(* Logix 5000 project; controller LeakTestAuto vendor 1 type 14 code 226 rev 37.11; software revision 37.01; part 6 of 15 *)

        [78].VolumeTest.Detailed.element_data[3].result_measurement := 5.014567, [78].LeakTest.Detailed.element_data[0].result_measurement := -999.0, [79].Barcode := 'A252620460', [79].VolumeTest.UID := 25864, [79].VolumeTest.Basic.unique_id := 25864, [79].VolumeTest.Basic.channel_num := 1, [79].VolumeTest.Basic.program_num := 1, [79].VolumeTest.Basic.evaluation_code := 2, [79].VolumeTest.Basic.test_port := 1, [79].VolumeTest.Basic.year := 26, [79].VolumeTest.Basic.month := 6, [79].VolumeTest.Basic.date := 2, [79].VolumeTest.Basic.hour := 14, [79].VolumeTest.Basic.minute := 38, [79].VolumeTest.Basic.second := 3, [79].VolumeTest.Basic.flags := 12, [79].VolumeTest.Basic.Num_tests := 1, [79].VolumeTest.Basic.test_elements.test_type := 69, [79].VolumeTest.Basic.test_elements.test_eval := 2, [79].VolumeTest.Basic.test_elements.num_elements := 4, [79].VolumeTest.Detailed.unique_id := 25864, [79].VolumeTest.Detailed.num_elements := 4, [79].VolumeTest.Detailed.Test_Type := 69, [79].VolumeTest.Detailed.element_data[0].Variable_code := 245, [79].VolumeTest.Detailed.element_data[0].prec_code := 2, [79].VolumeTest.Detailed.element_data[0].Unit_code := 165, [79].VolumeTest.Detailed.element_data[0].result_measurement := 214.08073, [79].VolumeTest.Detailed.element_data[1].Variable_code := 13, [79].VolumeTest.Detailed.element_data[1].prec_code := 3, [79].VolumeTest.Detailed.element_data[1].Unit_code := 12, [79].VolumeTest.Detailed.element_data[1].result_measurement := 1.5963289, [79].VolumeTest.Detailed.element_data[2].Variable_code := 247, [79].VolumeTest.Detailed.element_data[2].prec_code := 3, [79].VolumeTest.Detailed.element_data[2].Unit_code := 12, [79].VolumeTest.Detailed.element_data[2].result_measurement := 5.013761, [79].VolumeTest.Detailed.element_data[3].Variable_code := 295, [79].VolumeTest.Detailed.element_data[3].prec_code := 3, [79].VolumeTest.Detailed.element_data[3].Unit_code := 12, [79].VolumeTest.Detailed.element_data[3].result_measurement := 5.014567, [79].LeakTest.Detailed.element_data[0].result_measurement := -999.0, [80].Barcode := 'B252620568', [80].VolumeTest.UID := 26779, [80].VolumeTest.Basic.unique_id := 26779, [80].VolumeTest.Basic.channel_num := 1, [80].VolumeTest.Basic.program_num := 1, [80].VolumeTest.Basic.evaluation_code := 1, [80].VolumeTest.Basic.test_port := 1, [80].VolumeTest.Basic.year := 26, [80].VolumeTest.Basic.month := 6, [80].VolumeTest.Basic.date := 2, [80].VolumeTest.Basic.hour := 14, [80].VolumeTest.Basic.minute := 38, [80].VolumeTest.Basic.second := 48, [80].VolumeTest.Basic.flags := 12, [80].VolumeTest.Basic.Num_tests := 1, [80].VolumeTest.Basic.test_elements.test_type := 69, [80].VolumeTest.Basic.test_elements.test_eval := 1, [80].VolumeTest.Basic.test_elements.num_elements := 4, [80].VolumeTest.Detailed.unique_id := 26779, [80].VolumeTest.Detailed.num_elements := 4,
        [80].VolumeTest.Detailed.Test_Type := 69, [80].VolumeTest.Detailed.element_data[0].Variable_code := 245, [80].VolumeTest.Detailed.element_data[0].prec_code := 2, [80].VolumeTest.Detailed.element_data[0].Unit_code := 165, [80].VolumeTest.Detailed.element_data[0].result_measurement := 185.59888, [80].VolumeTest.Detailed.element_data[1].Variable_code := 13, [80].VolumeTest.Detailed.element_data[1].prec_code := 3, [80].VolumeTest.Detailed.element_data[1].Unit_code := 12, [80].VolumeTest.Detailed.element_data[1].result_measurement := 1.7575082, [80].VolumeTest.Detailed.element_data[2].Variable_code := 247, [80].VolumeTest.Detailed.element_data[2].prec_code := 3, [80].VolumeTest.Detailed.element_data[2].Unit_code := 12, [80].VolumeTest.Detailed.element_data[2].result_measurement := 5.0194235, [80].VolumeTest.Detailed.element_data[3].Variable_code := 295, [80].VolumeTest.Detailed.element_data[3].prec_code := 3, [80].VolumeTest.Detailed.element_data[3].Unit_code := 12, [80].VolumeTest.Detailed.element_data[3].result_measurement := 5.02042, [80].LeakTest.UID := 26780, [80].LeakTest.Basic.unique_id := 26780, [80].LeakTest.Basic.channel_num := 1, [80].LeakTest.Basic.program_num := 2, [80].LeakTest.Basic.evaluation_code := 1, [80].LeakTest.Basic.test_port := 1, [80].LeakTest.Basic.year := 26, [80].LeakTest.Basic.month := 6, [80].LeakTest.Basic.date := 2, [80].LeakTest.Basic.hour := 14, [80].LeakTest.Basic.minute := 38, [80].LeakTest.Basic.second := 54, [80].LeakTest.Basic.flags := 12, [80].LeakTest.Basic.Num_tests := 1, [80].LeakTest.Basic.test_elements.test_type := 66, [80].LeakTest.Basic.test_elements.test_eval := 1, [80].LeakTest.Basic.test_elements.num_elements := 16, [80].LeakTest.Detailed.unique_id := 26780, [80].LeakTest.Detailed.num_elements := 16, [80].LeakTest.Detailed.Test_Type := 66, [80].LeakTest.Detailed.element_data[0].Variable_code := 61, [80].LeakTest.Detailed.element_data[0].prec_code := 2, [80].LeakTest.Detailed.element_data[0].Unit_code := 60, [80].LeakTest.Detailed.element_data[0].result_measurement := -0.068731606, [80].LeakTest.Detailed.element_data[1].Variable_code := 28, [80].LeakTest.Detailed.element_data[1].prec_code := 3, [80].LeakTest.Detailed.element_data[1].Unit_code := 41, [80].LeakTest.Detailed.element_data[1].result_measurement := 0.0002514571, [80].LeakTest.Detailed.element_data[2].Variable_code := 13, [80].LeakTest.Detailed.element_data[2].prec_code := 3, [80].LeakTest.Detailed.element_data[2].Unit_code := 12, [80].LeakTest.Detailed.element_data[2].result_measurement := 5.0413327, [80].LeakTest.Detailed.element_data[3].Variable_code := 75, [80].LeakTest.Detailed.element_data[3].prec_code := 2, [80].LeakTest.Detailed.element_data[3].Unit_code := 60, [80].LeakTest.Detailed.element_data[4].Variable_code := 60, [80].LeakTest.Detailed.element_data[4].prec_code := 2, [80].LeakTest.Detailed.element_data[4].Unit_code := 60, [80].LeakTest.Detailed.element_data[4].result_measurement := -0.07878989, [80].LeakTest.Detailed.element_data[5].Variable_code := 56, [80].LeakTest.Detailed.element_data[5].prec_code := 3, [80].LeakTest.Detailed.element_data[5].Unit_code := 41, [80].LeakTest.Detailed.element_data[5].result_measurement := 0.00013038516,
        [80].LeakTest.Detailed.element_data[6].Variable_code := 55, [80].LeakTest.Detailed.element_data[6].prec_code := 3, [80].LeakTest.Detailed.element_data[6].Unit_code := 12, [80].LeakTest.Detailed.element_data[6].result_measurement := 5.0413327, [80].LeakTest.Detailed.element_data[7].Variable_code := 58, [80].LeakTest.Detailed.element_data[7].prec_code := 2, [80].LeakTest.Detailed.element_data[7].Unit_code := 60, [80].LeakTest.Detailed.element_data[7].result_measurement := -1.0002404, [80].LeakTest.Detailed.element_data[8].Variable_code := 59, [80].LeakTest.Detailed.element_data[8].prec_code := 2, [80].LeakTest.Detailed.element_data[8].Unit_code := 60, [80].LeakTest.Detailed.element_data[8].result_measurement := 1.0002404, [80].LeakTest.Detailed.element_data[9].Variable_code := 12, [80].LeakTest.Detailed.element_data[9].prec_code := 3, [80].LeakTest.Detailed.element_data[9].Unit_code := 12, [80].LeakTest.Detailed.element_data[9].result_measurement := 5.000001, [80].LeakTest.Detailed.element_data[10].Variable_code := 62, [80].LeakTest.Detailed.element_data[10].prec_code := 2, [80].LeakTest.Detailed.element_data[10].Unit_code := 60, [80].LeakTest.Detailed.element_data[10].result_measurement := 1.1002644, [80].LeakTest.Detailed.element_data[11].Variable_code := 21, [80].LeakTest.Detailed.element_data[11].prec_code := 3, [80].LeakTest.Detailed.element_data[11].Unit_code := 41, [80].LeakTest.Detailed.element_data[11].result_measurement := 0.0015180558, [80].LeakTest.Detailed.element_data[12].Variable_code := 25, [80].LeakTest.Detailed.element_data[12].prec_code := 3, [80].LeakTest.Detailed.element_data[12].Unit_code := 41, [80].LeakTest.Detailed.element_data[12].result_measurement := 0.021727756, [80].LeakTest.Detailed.element_data[13].Variable_code := 216, [80].LeakTest.Detailed.element_data[13].prec_code := 3, [80].LeakTest.Detailed.element_data[13].Unit_code := 41, [80].LeakTest.Detailed.element_data[13].result_measurement := 0.00085681677, [80].LeakTest.Detailed.element_data[14].Variable_code := 218, [80].LeakTest.Detailed.element_data[14].prec_code := 3, [80].LeakTest.Detailed.element_data[14].Unit_code := 41, [80].LeakTest.Detailed.element_data[14].result_measurement := 0.01094304, [80].LeakTest.Detailed.element_data[15].Variable_code := 295, [80].LeakTest.Detailed.element_data[15].prec_code := 3, [80].LeakTest.Detailed.element_data[15].Unit_code := 12, [80].LeakTest.Detailed.element_data[15].result_measurement := 5.04273, [81].Barcode := 'B252620571', [81].VolumeTest.UID := 26782, [81].VolumeTest.Basic.unique_id := 26782, [81].VolumeTest.Basic.channel_num := 1, [81].VolumeTest.Basic.program_num := 1, [81].VolumeTest.Basic.evaluation_code := 1, [81].VolumeTest.Basic.test_port := 1, [81].VolumeTest.Basic.year := 26, [81].VolumeTest.Basic.month := 6, [81].VolumeTest.Basic.date := 2, [81].VolumeTest.Basic.hour := 14, [81].VolumeTest.Basic.minute := 39, [81].VolumeTest.Basic.second := 10, [81].VolumeTest.Basic.flags := 12, [81].VolumeTest.Basic.Num_tests := 1, [81].VolumeTest.Basic.test_elements.test_type := 69, [81].VolumeTest.Basic.test_elements.test_eval := 1, [81].VolumeTest.Basic.test_elements.num_elements := 4, [81].VolumeTest.Detailed.unique_id := 26782, [81].VolumeTest.Detailed.num_elements := 4,
        [81].VolumeTest.Detailed.Test_Type := 69, [81].VolumeTest.Detailed.element_data[0].Variable_code := 245, [81].VolumeTest.Detailed.element_data[0].prec_code := 2, [81].VolumeTest.Detailed.element_data[0].Unit_code := 165, [81].VolumeTest.Detailed.element_data[0].result_measurement := 185.52951, [81].VolumeTest.Detailed.element_data[1].Variable_code := 13, [81].VolumeTest.Detailed.element_data[1].prec_code := 3, [81].VolumeTest.Detailed.element_data[1].Unit_code := 12, [81].VolumeTest.Detailed.element_data[1].result_measurement := 1.757997, [81].VolumeTest.Detailed.element_data[2].Variable_code := 247, [81].VolumeTest.Detailed.element_data[2].prec_code := 3, [81].VolumeTest.Detailed.element_data[2].Unit_code := 12, [81].VolumeTest.Detailed.element_data[2].result_measurement := 5.0196004, [81].VolumeTest.Detailed.element_data[3].Variable_code := 295, [81].VolumeTest.Detailed.element_data[3].prec_code := 3, [81].VolumeTest.Detailed.element_data[3].Unit_code := 12, [81].VolumeTest.Detailed.element_data[3].result_measurement := 5.0203876, [81].LeakTest.UID := 26783, [81].LeakTest.Basic.unique_id := 26783, [81].LeakTest.Basic.channel_num := 1, [81].LeakTest.Basic.program_num := 2, [81].LeakTest.Basic.evaluation_code := 1, [81].LeakTest.Basic.test_port := 1, [81].LeakTest.Basic.year := 26, [81].LeakTest.Basic.month := 6, [81].LeakTest.Basic.date := 2, [81].LeakTest.Basic.hour := 14, [81].LeakTest.Basic.minute := 39, [81].LeakTest.Basic.second := 17, [81].LeakTest.Basic.flags := 12, [81].LeakTest.Basic.Num_tests := 1, [81].LeakTest.Basic.test_elements.test_type := 66, [81].LeakTest.Basic.test_elements.test_eval := 1, [81].LeakTest.Basic.test_elements.num_elements := 16, [81].LeakTest.Detailed.unique_id := 26783, [81].LeakTest.Detailed.num_elements := 16, [81].LeakTest.Detailed.Test_Type := 66, [81].LeakTest.Detailed.element_data[0].Variable_code := 61, [81].LeakTest.Detailed.element_data[0].prec_code := 2, [81].LeakTest.Detailed.element_data[0].Unit_code := 60, [81].LeakTest.Detailed.element_data[0].result_measurement := -0.059232116, [81].LeakTest.Detailed.element_data[1].Variable_code := 28, [81].LeakTest.Detailed.element_data[1].prec_code := 3, [81].LeakTest.Detailed.element_data[1].Unit_code := 41, [81].LeakTest.Detailed.element_data[1].result_measurement := 0.00042840838, [81].LeakTest.Detailed.element_data[2].Variable_code := 13, [81].LeakTest.Detailed.element_data[2].prec_code := 3, [81].LeakTest.Detailed.element_data[2].Unit_code := 12, [81].LeakTest.Detailed.element_data[2].result_measurement := 5.040425, [81].LeakTest.Detailed.element_data[3].Variable_code := 75, [81].LeakTest.Detailed.element_data[3].prec_code := 2, [81].LeakTest.Detailed.element_data[3].Unit_code := 60, [81].LeakTest.Detailed.element_data[4].Variable_code := 60, [81].LeakTest.Detailed.element_data[4].prec_code := 2, [81].LeakTest.Detailed.element_data[4].Unit_code := 60, [81].LeakTest.Detailed.element_data[4].result_measurement := -0.068731606, [81].LeakTest.Detailed.element_data[5].Variable_code := 56, [81].LeakTest.Detailed.element_data[5].prec_code := 3, [81].LeakTest.Detailed.element_data[5].Unit_code := 41, [81].LeakTest.Detailed.element_data[5].result_measurement := 0.00022351742,
        [81].LeakTest.Detailed.element_data[6].Variable_code := 55, [81].LeakTest.Detailed.element_data[6].prec_code := 3, [81].LeakTest.Detailed.element_data[6].Unit_code := 12, [81].LeakTest.Detailed.element_data[6].result_measurement := 5.040425, [81].LeakTest.Detailed.element_data[7].Variable_code := 58, [81].LeakTest.Detailed.element_data[7].prec_code := 2, [81].LeakTest.Detailed.element_data[7].Unit_code := 60, [81].LeakTest.Detailed.element_data[7].result_measurement := -1.0002404, [81].LeakTest.Detailed.element_data[8].Variable_code := 59, [81].LeakTest.Detailed.element_data[8].prec_code := 2, [81].LeakTest.Detailed.element_data[8].Unit_code := 60, [81].LeakTest.Detailed.element_data[8].result_measurement := 1.0002404, [81].LeakTest.Detailed.element_data[9].Variable_code := 12, [81].LeakTest.Detailed.element_data[9].prec_code := 3, [81].LeakTest.Detailed.element_data[9].Unit_code := 12, [81].LeakTest.Detailed.element_data[9].result_measurement := 5.000001, [81].LeakTest.Detailed.element_data[10].Variable_code := 62, [81].LeakTest.Detailed.element_data[10].prec_code := 2, [81].LeakTest.Detailed.element_data[10].Unit_code := 60, [81].LeakTest.Detailed.element_data[10].result_measurement := 1.1002644, [81].LeakTest.Detailed.element_data[11].Variable_code := 21, [81].LeakTest.Detailed.element_data[11].prec_code := 3, [81].LeakTest.Detailed.element_data[11].Unit_code := 41, [81].LeakTest.Detailed.element_data[11].result_measurement := 0.0015180558, [81].LeakTest.Detailed.element_data[12].Variable_code := 25, [81].LeakTest.Detailed.element_data[12].prec_code := 3, [81].LeakTest.Detailed.element_data[12].Unit_code := 41, [81].LeakTest.Detailed.element_data[12].result_measurement := 0.021727756, [81].LeakTest.Detailed.element_data[13].Variable_code := 216, [81].LeakTest.Detailed.element_data[13].prec_code := 3, [81].LeakTest.Detailed.element_data[13].Unit_code := 41, [81].LeakTest.Detailed.element_data[13].result_measurement := 0.00085681677, [81].LeakTest.Detailed.element_data[14].Variable_code := 218, [81].LeakTest.Detailed.element_data[14].prec_code := 3, [81].LeakTest.Detailed.element_data[14].Unit_code := 41, [81].LeakTest.Detailed.element_data[14].result_measurement := 0.01094304, [81].LeakTest.Detailed.element_data[15].Variable_code := 295, [81].LeakTest.Detailed.element_data[15].prec_code := 3, [81].LeakTest.Detailed.element_data[15].Unit_code := 12, [81].LeakTest.Detailed.element_data[15].result_measurement := 5.0419664, [82].Barcode := 'B252620555', [82].VolumeTest.UID := 25866, [82].VolumeTest.Basic.unique_id := 25866, [82].VolumeTest.Basic.channel_num := 1, [82].VolumeTest.Basic.program_num := 1, [82].VolumeTest.Basic.evaluation_code := 1, [82].VolumeTest.Basic.test_port := 1, [82].VolumeTest.Basic.year := 26, [82].VolumeTest.Basic.month := 6, [82].VolumeTest.Basic.date := 2, [82].VolumeTest.Basic.hour := 14, [82].VolumeTest.Basic.minute := 38, [82].VolumeTest.Basic.second := 25, [82].VolumeTest.Basic.flags := 12, [82].VolumeTest.Basic.Num_tests := 1, [82].VolumeTest.Basic.test_elements.test_type := 69, [82].VolumeTest.Basic.test_elements.test_eval := 1, [82].VolumeTest.Basic.test_elements.num_elements := 4, [82].VolumeTest.Detailed.unique_id := 25866, [82].VolumeTest.Detailed.num_elements := 4,
        [82].VolumeTest.Detailed.Test_Type := 69, [82].VolumeTest.Detailed.element_data[0].Variable_code := 245, [82].VolumeTest.Detailed.element_data[0].prec_code := 2, [82].VolumeTest.Detailed.element_data[0].Unit_code := 165, [82].VolumeTest.Detailed.element_data[0].result_measurement := 188.30235, [82].VolumeTest.Detailed.element_data[1].Variable_code := 13, [82].VolumeTest.Detailed.element_data[1].prec_code := 3, [82].VolumeTest.Detailed.element_data[1].Unit_code := 12, [82].VolumeTest.Detailed.element_data[1].result_measurement := 1.7390168, [82].VolumeTest.Detailed.element_data[2].Variable_code := 247, [82].VolumeTest.Detailed.element_data[2].prec_code := 3, [82].VolumeTest.Detailed.element_data[2].Unit_code := 12, [82].VolumeTest.Detailed.element_data[2].result_measurement := 5.013626, [82].VolumeTest.Detailed.element_data[3].Variable_code := 295, [82].VolumeTest.Detailed.element_data[3].prec_code := 3, [82].VolumeTest.Detailed.element_data[3].Unit_code := 12, [82].VolumeTest.Detailed.element_data[3].result_measurement := 5.0143385, [82].LeakTest.UID := 25867, [82].LeakTest.Basic.unique_id := 25867, [82].LeakTest.Basic.channel_num := 1, [82].LeakTest.Basic.program_num := 2, [82].LeakTest.Basic.evaluation_code := 1, [82].LeakTest.Basic.test_port := 1, [82].LeakTest.Basic.year := 26, [82].LeakTest.Basic.month := 6, [82].LeakTest.Basic.date := 2, [82].LeakTest.Basic.hour := 14, [82].LeakTest.Basic.minute := 38, [82].LeakTest.Basic.second := 32, [82].LeakTest.Basic.flags := 12, [82].LeakTest.Basic.Num_tests := 1, [82].LeakTest.Basic.test_elements.test_type := 66, [82].LeakTest.Basic.test_elements.test_eval := 1, [82].LeakTest.Basic.test_elements.num_elements := 16, [82].LeakTest.Detailed.unique_id := 25867, [82].LeakTest.Detailed.num_elements := 16, [82].LeakTest.Detailed.Test_Type := 66, [82].LeakTest.Detailed.element_data[0].Variable_code := 61, [82].LeakTest.Detailed.element_data[0].prec_code := 2, [82].LeakTest.Detailed.element_data[0].Unit_code := 60, [82].LeakTest.Detailed.element_data[0].result_measurement := -0.05811453, [82].LeakTest.Detailed.element_data[1].Variable_code := 28, [82].LeakTest.Detailed.element_data[1].prec_code := 3, [82].LeakTest.Detailed.element_data[1].Unit_code := 41, [82].LeakTest.Detailed.element_data[1].result_measurement := 0.00045634806, [82].LeakTest.Detailed.element_data[2].Variable_code := 13, [82].LeakTest.Detailed.element_data[2].prec_code := 3, [82].LeakTest.Detailed.element_data[2].Unit_code := 12, [82].LeakTest.Detailed.element_data[2].result_measurement := 5.033845, [82].LeakTest.Detailed.element_data[3].Variable_code := 75, [82].LeakTest.Detailed.element_data[3].prec_code := 2, [82].LeakTest.Detailed.element_data[3].Unit_code := 60, [82].LeakTest.Detailed.element_data[4].Variable_code := 60, [82].LeakTest.Detailed.element_data[4].prec_code := 2, [82].LeakTest.Detailed.element_data[4].Unit_code := 60, [82].LeakTest.Detailed.element_data[4].result_measurement := -0.07431954, [82].LeakTest.Detailed.element_data[5].Variable_code := 56, [82].LeakTest.Detailed.element_data[5].prec_code := 3, [82].LeakTest.Detailed.element_data[5].Unit_code := 41, [82].LeakTest.Detailed.element_data[5].result_measurement := 0.00017695129,
        [82].LeakTest.Detailed.element_data[6].Variable_code := 55, [82].LeakTest.Detailed.element_data[6].prec_code := 3, [82].LeakTest.Detailed.element_data[6].Unit_code := 12, [82].LeakTest.Detailed.element_data[6].result_measurement := 5.033845, [82].LeakTest.Detailed.element_data[7].Variable_code := 58, [82].LeakTest.Detailed.element_data[7].prec_code := 2, [82].LeakTest.Detailed.element_data[7].Unit_code := 60, [82].LeakTest.Detailed.element_data[7].result_measurement := -1.0002404, [82].LeakTest.Detailed.element_data[8].Variable_code := 59, [82].LeakTest.Detailed.element_data[8].prec_code := 2, [82].LeakTest.Detailed.element_data[8].Unit_code := 60, [82].LeakTest.Detailed.element_data[8].result_measurement := 1.0002404, [82].LeakTest.Detailed.element_data[9].Variable_code := 12, [82].LeakTest.Detailed.element_data[9].prec_code := 3, [82].LeakTest.Detailed.element_data[9].Unit_code := 12, [82].LeakTest.Detailed.element_data[9].result_measurement := 5.000001, [82].LeakTest.Detailed.element_data[10].Variable_code := 62, [82].LeakTest.Detailed.element_data[10].prec_code := 2, [82].LeakTest.Detailed.element_data[10].Unit_code := 60, [82].LeakTest.Detailed.element_data[10].result_measurement := 1.109764, [82].LeakTest.Detailed.element_data[11].Variable_code := 21, [82].LeakTest.Detailed.element_data[11].prec_code := 3, [82].LeakTest.Detailed.element_data[11].Unit_code := 41, [82].LeakTest.Detailed.element_data[11].result_measurement := 0.0015180558, [82].LeakTest.Detailed.element_data[12].Variable_code := 25, [82].LeakTest.Detailed.element_data[12].prec_code := 3, [82].LeakTest.Detailed.element_data[12].Unit_code := 41, [82].LeakTest.Detailed.element_data[12].result_measurement := 0.021727756, [82].LeakTest.Detailed.element_data[13].Variable_code := 216, [82].LeakTest.Detailed.element_data[13].prec_code := 3, [82].LeakTest.Detailed.element_data[13].Unit_code := 41, [82].LeakTest.Detailed.element_data[13].result_measurement := 0.00085681677, [82].LeakTest.Detailed.element_data[14].Variable_code := 218, [82].LeakTest.Detailed.element_data[14].prec_code := 3, [82].LeakTest.Detailed.element_data[14].Unit_code := 41, [82].LeakTest.Detailed.element_data[14].result_measurement := 0.01094304, [82].LeakTest.Detailed.element_data[15].Variable_code := 295, [82].LeakTest.Detailed.element_data[15].prec_code := 3, [82].LeakTest.Detailed.element_data[15].Unit_code := 12, [82].LeakTest.Detailed.element_data[15].result_measurement := 5.03602, [83].Barcode := 'B252620555', [83].VolumeTest.UID := 41945, [83].VolumeTest.Basic.unique_id := 41945, [83].VolumeTest.Basic.channel_num := 1, [83].VolumeTest.Basic.program_num := 1, [83].VolumeTest.Basic.evaluation_code := 1, [83].VolumeTest.Basic.test_port := 1, [83].VolumeTest.Basic.year := 26, [83].VolumeTest.Basic.month := 6, [83].VolumeTest.Basic.date := 4, [83].VolumeTest.Basic.hour := 12, [83].VolumeTest.Basic.minute := 27, [83].VolumeTest.Basic.second := 3, [83].VolumeTest.Basic.flags := 12, [83].VolumeTest.Basic.Num_tests := 1, [83].VolumeTest.Basic.test_elements.test_type := 69, [83].VolumeTest.Basic.test_elements.test_eval := 1, [83].VolumeTest.Basic.test_elements.num_elements := 4, [83].VolumeTest.Detailed.unique_id := 41945, [83].VolumeTest.Detailed.num_elements := 4,
        [83].VolumeTest.Detailed.Test_Type := 69, [83].VolumeTest.Detailed.element_data[0].Variable_code := 245, [83].VolumeTest.Detailed.element_data[0].prec_code := 2, [83].VolumeTest.Detailed.element_data[0].Unit_code := 165, [83].VolumeTest.Detailed.element_data[0].result_measurement := 186.67934, [83].VolumeTest.Detailed.element_data[1].Variable_code := 13, [83].VolumeTest.Detailed.element_data[1].prec_code := 3, [83].VolumeTest.Detailed.element_data[1].Unit_code := 12, [83].VolumeTest.Detailed.element_data[1].result_measurement := 1.7815549, [83].VolumeTest.Detailed.element_data[2].Variable_code := 247, [83].VolumeTest.Detailed.element_data[2].prec_code := 3, [83].VolumeTest.Detailed.element_data[2].Unit_code := 12, [83].VolumeTest.Detailed.element_data[2].result_measurement := 5.10735, [83].VolumeTest.Detailed.element_data[3].Variable_code := 295, [83].VolumeTest.Detailed.element_data[3].prec_code := 3, [83].VolumeTest.Detailed.element_data[3].Unit_code := 12, [83].VolumeTest.Detailed.element_data[3].result_measurement := 5.107876, [83].LeakTest.UID := 41946, [83].LeakTest.Basic.unique_id := 41946, [83].LeakTest.Basic.channel_num := 1, [83].LeakTest.Basic.program_num := 2, [83].LeakTest.Basic.evaluation_code := 1, [83].LeakTest.Basic.test_port := 1, [83].LeakTest.Basic.year := 26, [83].LeakTest.Basic.month := 6, [83].LeakTest.Basic.date := 4, [83].LeakTest.Basic.hour := 12, [83].LeakTest.Basic.minute := 27, [83].LeakTest.Basic.second := 10, [83].LeakTest.Basic.flags := 12, [83].LeakTest.Basic.Num_tests := 1, [83].LeakTest.Basic.test_elements.test_type := 66, [83].LeakTest.Basic.test_elements.test_eval := 1, [83].LeakTest.Basic.test_elements.num_elements := 16, [83].LeakTest.Detailed.unique_id := 41946, [83].LeakTest.Detailed.num_elements := 16, [83].LeakTest.Detailed.Test_Type := 66, [83].LeakTest.Detailed.element_data[0].Variable_code := 61, [83].LeakTest.Detailed.element_data[0].prec_code := 2, [83].LeakTest.Detailed.element_data[0].Unit_code := 60, [83].LeakTest.Detailed.element_data[0].result_measurement := -0.07431954, [83].LeakTest.Detailed.element_data[1].Variable_code := 28, [83].LeakTest.Detailed.element_data[1].prec_code := 3, [83].LeakTest.Detailed.element_data[1].Unit_code := 41, [83].LeakTest.Detailed.element_data[1].result_measurement := 0.00014901161, [83].LeakTest.Detailed.element_data[2].Variable_code := 13, [83].LeakTest.Detailed.element_data[2].prec_code := 3, [83].LeakTest.Detailed.element_data[2].Unit_code := 12, [83].LeakTest.Detailed.element_data[2].result_measurement := 5.137217, [83].LeakTest.Detailed.element_data[3].Variable_code := 75, [83].LeakTest.Detailed.element_data[3].prec_code := 2, [83].LeakTest.Detailed.element_data[3].Unit_code := 60, [83].LeakTest.Detailed.element_data[4].Variable_code := 60, [83].LeakTest.Detailed.element_data[4].prec_code := 2, [83].LeakTest.Detailed.element_data[4].Unit_code := 60, [83].LeakTest.Detailed.element_data[4].result_measurement := -0.08214265, [83].LeakTest.Detailed.element_data[5].Variable_code := 56, [83].LeakTest.Detailed.element_data[5].prec_code := 3, [83].LeakTest.Detailed.element_data[5].Unit_code := 41, [83].LeakTest.Detailed.element_data[5].result_measurement := 0.00010244548,
        [83].LeakTest.Detailed.element_data[6].Variable_code := 55, [83].LeakTest.Detailed.element_data[6].prec_code := 3, [83].LeakTest.Detailed.element_data[6].Unit_code := 12, [83].LeakTest.Detailed.element_data[6].result_measurement := 5.137217, [83].LeakTest.Detailed.element_data[7].Variable_code := 58, [83].LeakTest.Detailed.element_data[7].prec_code := 2, [83].LeakTest.Detailed.element_data[7].Unit_code := 60, [83].LeakTest.Detailed.element_data[7].result_measurement := -1.0002404, [83].LeakTest.Detailed.element_data[8].Variable_code := 59, [83].LeakTest.Detailed.element_data[8].prec_code := 2, [83].LeakTest.Detailed.element_data[8].Unit_code := 60, [83].LeakTest.Detailed.element_data[8].result_measurement := 1.0002404, [83].LeakTest.Detailed.element_data[9].Variable_code := 12, [83].LeakTest.Detailed.element_data[9].prec_code := 3, [83].LeakTest.Detailed.element_data[9].Unit_code := 12, [83].LeakTest.Detailed.element_data[9].result_measurement := 5.000001, [83].LeakTest.Detailed.element_data[10].Variable_code := 62, [83].LeakTest.Detailed.element_data[10].prec_code := 2, [83].LeakTest.Detailed.element_data[10].Unit_code := 60, [83].LeakTest.Detailed.element_data[10].result_measurement := 1.1002644, [83].LeakTest.Detailed.element_data[11].Variable_code := 21, [83].LeakTest.Detailed.element_data[11].prec_code := 3, [83].LeakTest.Detailed.element_data[11].Unit_code := 41, [83].LeakTest.Detailed.element_data[11].result_measurement := 0.0015180558, [83].LeakTest.Detailed.element_data[12].Variable_code := 25, [83].LeakTest.Detailed.element_data[12].prec_code := 3, [83].LeakTest.Detailed.element_data[12].Unit_code := 41, [83].LeakTest.Detailed.element_data[12].result_measurement := 0.021727756, [83].LeakTest.Detailed.element_data[13].Variable_code := 216, [83].LeakTest.Detailed.element_data[13].prec_code := 3, [83].LeakTest.Detailed.element_data[13].Unit_code := 41, [83].LeakTest.Detailed.element_data[13].result_measurement := 0.00085681677, [83].LeakTest.Detailed.element_data[14].Variable_code := 218, [83].LeakTest.Detailed.element_data[14].prec_code := 3, [83].LeakTest.Detailed.element_data[14].Unit_code := 41, [83].LeakTest.Detailed.element_data[14].result_measurement := 0.01094304, [83].LeakTest.Detailed.element_data[15].Variable_code := 295, [83].LeakTest.Detailed.element_data[15].prec_code := 3, [83].LeakTest.Detailed.element_data[15].Unit_code := 12, [83].LeakTest.Detailed.element_data[15].result_measurement := 5.1387258, [84].Barcode := 'B252620571', [84].VolumeTest.UID := 42936, [84].VolumeTest.Basic.unique_id := 42936, [84].VolumeTest.Basic.channel_num := 1, [84].VolumeTest.Basic.program_num := 1, [84].VolumeTest.Basic.evaluation_code := 1, [84].VolumeTest.Basic.test_port := 1, [84].VolumeTest.Basic.year := 26, [84].VolumeTest.Basic.month := 6, [84].VolumeTest.Basic.date := 4, [84].VolumeTest.Basic.hour := 12, [84].VolumeTest.Basic.minute := 27, [84].VolumeTest.Basic.second := 27, [84].VolumeTest.Basic.flags := 12, [84].VolumeTest.Basic.Num_tests := 1, [84].VolumeTest.Basic.test_elements.test_type := 69, [84].VolumeTest.Basic.test_elements.test_eval := 1, [84].VolumeTest.Basic.test_elements.num_elements := 4, [84].VolumeTest.Detailed.unique_id := 42936, [84].VolumeTest.Detailed.num_elements := 4,
        [84].VolumeTest.Detailed.Test_Type := 69, [84].VolumeTest.Detailed.element_data[0].Variable_code := 245, [84].VolumeTest.Detailed.element_data[0].prec_code := 2, [84].VolumeTest.Detailed.element_data[0].Unit_code := 165, [84].VolumeTest.Detailed.element_data[0].result_measurement := 188.14069, [84].VolumeTest.Detailed.element_data[1].Variable_code := 13, [84].VolumeTest.Detailed.element_data[1].prec_code := 3, [84].VolumeTest.Detailed.element_data[1].Unit_code := 12, [84].VolumeTest.Detailed.element_data[1].result_measurement := 1.8124143, [84].VolumeTest.Detailed.element_data[2].Variable_code := 247, [84].VolumeTest.Detailed.element_data[2].prec_code := 3, [84].VolumeTest.Detailed.element_data[2].Unit_code := 12, [84].VolumeTest.Detailed.element_data[2].result_measurement := 5.222303, [84].VolumeTest.Detailed.element_data[3].Variable_code := 295, [84].VolumeTest.Detailed.element_data[3].prec_code := 3, [84].VolumeTest.Detailed.element_data[3].Unit_code := 12, [84].VolumeTest.Detailed.element_data[3].result_measurement := 5.224529, [84].LeakTest.UID := 42937, [84].LeakTest.Basic.unique_id := 42937, [84].LeakTest.Basic.channel_num := 1, [84].LeakTest.Basic.program_num := 2, [84].LeakTest.Basic.evaluation_code := 1, [84].LeakTest.Basic.test_port := 1, [84].LeakTest.Basic.year := 26, [84].LeakTest.Basic.month := 6, [84].LeakTest.Basic.date := 4, [84].LeakTest.Basic.hour := 12, [84].LeakTest.Basic.minute := 27, [84].LeakTest.Basic.second := 33, [84].LeakTest.Basic.flags := 12, [84].LeakTest.Basic.Num_tests := 1, [84].LeakTest.Basic.test_elements.test_type := 66, [84].LeakTest.Basic.test_elements.test_eval := 1, [84].LeakTest.Basic.test_elements.num_elements := 16, [84].LeakTest.Detailed.unique_id := 42937, [84].LeakTest.Detailed.num_elements := 16, [84].LeakTest.Detailed.Test_Type := 66, [84].LeakTest.Detailed.element_data[0].Variable_code := 61, [84].LeakTest.Detailed.element_data[0].prec_code := 2, [84].LeakTest.Detailed.element_data[0].Unit_code := 60, [84].LeakTest.Detailed.element_data[0].result_measurement := -0.005029142, [84].LeakTest.Detailed.element_data[1].Variable_code := 28, [84].LeakTest.Detailed.element_data[1].prec_code := 3, [84].LeakTest.Detailed.element_data[1].Unit_code := 41, [84].LeakTest.Detailed.element_data[1].result_measurement := -0.00010244548, [84].LeakTest.Detailed.element_data[2].Variable_code := 13, [84].LeakTest.Detailed.element_data[2].prec_code := 3, [84].LeakTest.Detailed.element_data[2].Unit_code := 12, [84].LeakTest.Detailed.element_data[2].result_measurement := 5.2362356, [84].LeakTest.Detailed.element_data[3].Variable_code := 75, [84].LeakTest.Detailed.element_data[3].prec_code := 2, [84].LeakTest.Detailed.element_data[3].Unit_code := 60, [84].LeakTest.Detailed.element_data[4].Variable_code := 60, [84].LeakTest.Detailed.element_data[4].prec_code := 2, [84].LeakTest.Detailed.element_data[4].Unit_code := 60, [84].LeakTest.Detailed.element_data[4].result_measurement := -0.022910535, [84].LeakTest.Detailed.element_data[5].Variable_code := 56, [84].LeakTest.Detailed.element_data[5].prec_code := 3, [84].LeakTest.Detailed.element_data[5].Unit_code := 41, [84].LeakTest.Detailed.element_data[5].result_measurement := -0.00027474016,
        [84].LeakTest.Detailed.element_data[6].Variable_code := 55, [84].LeakTest.Detailed.element_data[6].prec_code := 3, [84].LeakTest.Detailed.element_data[6].Unit_code := 12, [84].LeakTest.Detailed.element_data[6].result_measurement := 5.2362356, [84].LeakTest.Detailed.element_data[7].Variable_code := 58, [84].LeakTest.Detailed.element_data[7].prec_code := 2, [84].LeakTest.Detailed.element_data[7].Unit_code := 60, [84].LeakTest.Detailed.element_data[7].result_measurement := -1.0002404, [84].LeakTest.Detailed.element_data[8].Variable_code := 59, [84].LeakTest.Detailed.element_data[8].prec_code := 2, [84].LeakTest.Detailed.element_data[8].Unit_code := 60, [84].LeakTest.Detailed.element_data[8].result_measurement := 1.0002404, [84].LeakTest.Detailed.element_data[9].Variable_code := 12, [84].LeakTest.Detailed.element_data[9].prec_code := 3, [84].LeakTest.Detailed.element_data[9].Unit_code := 12, [84].LeakTest.Detailed.element_data[9].result_measurement := 5.000001, [84].LeakTest.Detailed.element_data[10].Variable_code := 62, [84].LeakTest.Detailed.element_data[10].prec_code := 2, [84].LeakTest.Detailed.element_data[10].Unit_code := 60, [84].LeakTest.Detailed.element_data[10].result_measurement := 1.1298805, [84].LeakTest.Detailed.element_data[11].Variable_code := 21, [84].LeakTest.Detailed.element_data[11].prec_code := 3, [84].LeakTest.Detailed.element_data[11].Unit_code := 41, [84].LeakTest.Detailed.element_data[11].result_measurement := 4.656613e-06, [84].LeakTest.Detailed.element_data[12].Variable_code := 25, [84].LeakTest.Detailed.element_data[12].prec_code := 3, [84].LeakTest.Detailed.element_data[12].Unit_code := 41, [84].LeakTest.Detailed.element_data[12].result_measurement := 0.023245811, [84].LeakTest.Detailed.element_data[13].Variable_code := 216, [84].LeakTest.Detailed.element_data[13].prec_code := 3, [84].LeakTest.Detailed.element_data[13].Unit_code := 41, [84].LeakTest.Detailed.element_data[13].result_measurement := -3.7252903e-05, [84].LeakTest.Detailed.element_data[14].Variable_code := 218, [84].LeakTest.Detailed.element_data[14].prec_code := 3, [84].LeakTest.Detailed.element_data[14].Unit_code := 41, [84].LeakTest.Detailed.element_data[14].result_measurement := 0.011632219, [84].LeakTest.Detailed.element_data[15].Variable_code := 295, [84].LeakTest.Detailed.element_data[15].prec_code := 3, [84].LeakTest.Detailed.element_data[15].Unit_code := 12, [84].LeakTest.Detailed.element_data[15].result_measurement := 5.237949, [85].Barcode := 'B252620865', [85].VolumeTest.UID := 42939, [85].VolumeTest.Basic.unique_id := 42939, [85].VolumeTest.Basic.channel_num := 1, [85].VolumeTest.Basic.program_num := 1, [85].VolumeTest.Basic.evaluation_code := 1, [85].VolumeTest.Basic.test_port := 1, [85].VolumeTest.Basic.year := 26, [85].VolumeTest.Basic.month := 6, [85].VolumeTest.Basic.date := 4, [85].VolumeTest.Basic.hour := 12, [85].VolumeTest.Basic.minute := 28, [85].VolumeTest.Basic.second := 27, [85].VolumeTest.Basic.flags := 12, [85].VolumeTest.Basic.Num_tests := 1, [85].VolumeTest.Basic.test_elements.test_type := 69, [85].VolumeTest.Basic.test_elements.test_eval := 1, [85].VolumeTest.Basic.test_elements.num_elements := 4, [85].VolumeTest.Detailed.unique_id := 42939, [85].VolumeTest.Detailed.num_elements := 4,
        [85].VolumeTest.Detailed.Test_Type := 69, [85].VolumeTest.Detailed.element_data[0].Variable_code := 245, [85].VolumeTest.Detailed.element_data[0].prec_code := 2, [85].VolumeTest.Detailed.element_data[0].Unit_code := 165, [85].VolumeTest.Detailed.element_data[0].result_measurement := 188.86253, [85].VolumeTest.Detailed.element_data[1].Variable_code := 13, [85].VolumeTest.Detailed.element_data[1].prec_code := 3, [85].VolumeTest.Detailed.element_data[1].Unit_code := 12, [85].VolumeTest.Detailed.element_data[1].result_measurement := 1.8058717, [85].VolumeTest.Detailed.element_data[2].Variable_code := 247, [85].VolumeTest.Detailed.element_data[2].prec_code := 3, [85].VolumeTest.Detailed.element_data[2].Unit_code := 12, [85].VolumeTest.Detailed.element_data[2].result_measurement := 5.216487, [85].VolumeTest.Detailed.element_data[3].Variable_code := 295, [85].VolumeTest.Detailed.element_data[3].prec_code := 3, [85].VolumeTest.Detailed.element_data[3].Unit_code := 12, [85].VolumeTest.Detailed.element_data[3].result_measurement := 5.2191176, [85].LeakTest.UID := 42940, [85].LeakTest.Basic.unique_id := 42940, [85].LeakTest.Basic.channel_num := 1, [85].LeakTest.Basic.program_num := 2, [85].LeakTest.Basic.evaluation_code := 1, [85].LeakTest.Basic.test_port := 1, [85].LeakTest.Basic.year := 26, [85].LeakTest.Basic.month := 6, [85].LeakTest.Basic.date := 4, [85].LeakTest.Basic.hour := 12, [85].LeakTest.Basic.minute := 28, [85].LeakTest.Basic.second := 34, [85].LeakTest.Basic.flags := 12, [85].LeakTest.Basic.Num_tests := 1, [85].LeakTest.Basic.test_elements.test_type := 66, [85].LeakTest.Basic.test_elements.test_eval := 1, [85].LeakTest.Basic.test_elements.num_elements := 16, [85].LeakTest.Detailed.unique_id := 42940, [85].LeakTest.Detailed.num_elements := 16, [85].LeakTest.Detailed.Test_Type := 66, [85].LeakTest.Detailed.element_data[0].Variable_code := 61, [85].LeakTest.Detailed.element_data[0].prec_code := 2, [85].LeakTest.Detailed.element_data[0].Unit_code := 60, [85].LeakTest.Detailed.element_data[0].result_measurement := -0.0067055225, [85].LeakTest.Detailed.element_data[1].Variable_code := 28, [85].LeakTest.Detailed.element_data[1].prec_code := 3, [85].LeakTest.Detailed.element_data[1].Unit_code := 41, [85].LeakTest.Detailed.element_data[1].result_measurement := -0.00013969839, [85].LeakTest.Detailed.element_data[2].Variable_code := 13, [85].LeakTest.Detailed.element_data[2].prec_code := 3, [85].LeakTest.Detailed.element_data[2].Unit_code := 12, [85].LeakTest.Detailed.element_data[2].result_measurement := 5.2345915, [85].LeakTest.Detailed.element_data[3].Variable_code := 75, [85].LeakTest.Detailed.element_data[3].prec_code := 2, [85].LeakTest.Detailed.element_data[3].Unit_code := 60, [85].LeakTest.Detailed.element_data[4].Variable_code := 60, [85].LeakTest.Detailed.element_data[4].prec_code := 2, [85].LeakTest.Detailed.element_data[4].Unit_code := 60, [85].LeakTest.Detailed.element_data[4].result_measurement := -0.0044703484, [85].LeakTest.Detailed.element_data[5].Variable_code := 56, [85].LeakTest.Detailed.element_data[5].prec_code := 3, [85].LeakTest.Detailed.element_data[5].Unit_code := 41, [85].LeakTest.Detailed.element_data[5].result_measurement := -8.8475645e-05,
        [85].LeakTest.Detailed.element_data[6].Variable_code := 55, [85].LeakTest.Detailed.element_data[6].prec_code := 3, [85].LeakTest.Detailed.element_data[6].Unit_code := 12, [85].LeakTest.Detailed.element_data[6].result_measurement := 5.2345915, [85].LeakTest.Detailed.element_data[7].Variable_code := 58, [85].LeakTest.Detailed.element_data[7].prec_code := 2, [85].LeakTest.Detailed.element_data[7].Unit_code := 60, [85].LeakTest.Detailed.element_data[7].result_measurement := -1.0002404, [85].LeakTest.Detailed.element_data[8].Variable_code := 59, [85].LeakTest.Detailed.element_data[8].prec_code := 2, [85].LeakTest.Detailed.element_data[8].Unit_code := 60, [85].LeakTest.Detailed.element_data[8].result_measurement := 1.0002404, [85].LeakTest.Detailed.element_data[9].Variable_code := 12, [85].LeakTest.Detailed.element_data[9].prec_code := 3, [85].LeakTest.Detailed.element_data[9].Unit_code := 12, [85].LeakTest.Detailed.element_data[9].result_measurement := 5.000001, [85].LeakTest.Detailed.element_data[10].Variable_code := 62, [85].LeakTest.Detailed.element_data[10].prec_code := 2, [85].LeakTest.Detailed.element_data[10].Unit_code := 60, [85].LeakTest.Detailed.element_data[10].result_measurement := 1.1298805, [85].LeakTest.Detailed.element_data[11].Variable_code := 21, [85].LeakTest.Detailed.element_data[11].prec_code := 3, [85].LeakTest.Detailed.element_data[11].Unit_code := 41, [85].LeakTest.Detailed.element_data[11].result_measurement := 4.656613e-06, [85].LeakTest.Detailed.element_data[12].Variable_code := 25, [85].LeakTest.Detailed.element_data[12].prec_code := 3, [85].LeakTest.Detailed.element_data[12].Unit_code := 41, [85].LeakTest.Detailed.element_data[12].result_measurement := 0.023245811, [85].LeakTest.Detailed.element_data[13].Variable_code := 216, [85].LeakTest.Detailed.element_data[13].prec_code := 3, [85].LeakTest.Detailed.element_data[13].Unit_code := 41, [85].LeakTest.Detailed.element_data[13].result_measurement := -3.7252903e-05, [85].LeakTest.Detailed.element_data[14].Variable_code := 218, [85].LeakTest.Detailed.element_data[14].prec_code := 3, [85].LeakTest.Detailed.element_data[14].Unit_code := 41, [85].LeakTest.Detailed.element_data[14].result_measurement := 0.011632219, [85].LeakTest.Detailed.element_data[15].Variable_code := 295, [85].LeakTest.Detailed.element_data[15].prec_code := 3, [85].LeakTest.Detailed.element_data[15].Unit_code := 12, [85].LeakTest.Detailed.element_data[15].result_measurement := 5.236021, [86].Barcode := 'B252620863', [86].VolumeTest.UID := 42946, [86].VolumeTest.Basic.unique_id := 42946, [86].VolumeTest.Basic.channel_num := 1, [86].VolumeTest.Basic.program_num := 1, [86].VolumeTest.Basic.evaluation_code := 1, [86].VolumeTest.Basic.test_port := 1, [86].VolumeTest.Basic.year := 26, [86].VolumeTest.Basic.month := 6, [86].VolumeTest.Basic.date := 4, [86].VolumeTest.Basic.hour := 14, [86].VolumeTest.Basic.minute := 58, [86].VolumeTest.Basic.second := 38, [86].VolumeTest.Basic.flags := 12, [86].VolumeTest.Basic.Num_tests := 1, [86].VolumeTest.Basic.test_elements.test_type := 69, [86].VolumeTest.Basic.test_elements.test_eval := 1, [86].VolumeTest.Basic.test_elements.num_elements := 4, [86].VolumeTest.Detailed.unique_id := 42946, [86].VolumeTest.Detailed.num_elements := 4,
        [86].VolumeTest.Detailed.Test_Type := 69, [86].VolumeTest.Detailed.element_data[0].Variable_code := 245, [86].VolumeTest.Detailed.element_data[0].prec_code := 2, [86].VolumeTest.Detailed.element_data[0].Unit_code := 165, [86].VolumeTest.Detailed.element_data[0].result_measurement := 188.01074, [86].VolumeTest.Detailed.element_data[1].Variable_code := 13, [86].VolumeTest.Detailed.element_data[1].prec_code := 3, [86].VolumeTest.Detailed.element_data[1].Unit_code := 12, [86].VolumeTest.Detailed.element_data[1].result_measurement := 1.8123071, [86].VolumeTest.Detailed.element_data[2].Variable_code := 247, [86].VolumeTest.Detailed.element_data[2].prec_code := 3, [86].VolumeTest.Detailed.element_data[2].Unit_code := 12, [86].VolumeTest.Detailed.element_data[2].result_measurement := 5.2196393, [86].VolumeTest.Detailed.element_data[3].Variable_code := 295, [86].VolumeTest.Detailed.element_data[3].prec_code := 3, [86].VolumeTest.Detailed.element_data[3].Unit_code := 12, [86].VolumeTest.Detailed.element_data[3].result_measurement := 5.220268, [86].LeakTest.UID := 42947, [86].LeakTest.Basic.unique_id := 42947, [86].LeakTest.Basic.channel_num := 1, [86].LeakTest.Basic.program_num := 2, [86].LeakTest.Basic.evaluation_code := 1, [86].LeakTest.Basic.test_port := 1, [86].LeakTest.Basic.year := 26, [86].LeakTest.Basic.month := 6, [86].LeakTest.Basic.date := 4, [86].LeakTest.Basic.hour := 14, [86].LeakTest.Basic.minute := 58, [86].LeakTest.Basic.second := 45, [86].LeakTest.Basic.flags := 12, [86].LeakTest.Basic.Num_tests := 1, [86].LeakTest.Basic.test_elements.test_type := 66, [86].LeakTest.Basic.test_elements.test_eval := 1, [86].LeakTest.Basic.test_elements.num_elements := 16, [86].LeakTest.Detailed.unique_id := 42947, [86].LeakTest.Detailed.num_elements := 16, [86].LeakTest.Detailed.Test_Type := 66, [86].LeakTest.Detailed.element_data[0].Variable_code := 61, [86].LeakTest.Detailed.element_data[0].prec_code := 2, [86].LeakTest.Detailed.element_data[0].Unit_code := 60, [86].LeakTest.Detailed.element_data[0].result_measurement := 0.00055879354, [86].LeakTest.Detailed.element_data[1].Variable_code := 28, [86].LeakTest.Detailed.element_data[1].prec_code := 3, [86].LeakTest.Detailed.element_data[1].Unit_code := 41, [86].LeakTest.Detailed.element_data[1].result_measurement := 1.8626451e-05, [86].LeakTest.Detailed.element_data[2].Variable_code := 13, [86].LeakTest.Detailed.element_data[2].prec_code := 3, [86].LeakTest.Detailed.element_data[2].Unit_code := 12, [86].LeakTest.Detailed.element_data[2].result_measurement := 5.2330036, [86].LeakTest.Detailed.element_data[3].Variable_code := 75, [86].LeakTest.Detailed.element_data[3].prec_code := 2, [86].LeakTest.Detailed.element_data[3].Unit_code := 60, [86].LeakTest.Detailed.element_data[4].Variable_code := 60, [86].LeakTest.Detailed.element_data[4].prec_code := 2, [86].LeakTest.Detailed.element_data[4].Unit_code := 60, [86].LeakTest.Detailed.element_data[4].result_measurement := 0.0067055225, [86].LeakTest.Detailed.element_data[5].Variable_code := 56, [86].LeakTest.Detailed.element_data[5].prec_code := 3, [86].LeakTest.Detailed.element_data[5].Unit_code := 41, [86].LeakTest.Detailed.element_data[5].result_measurement := 3.7252903e-05,
        [86].LeakTest.Detailed.element_data[6].Variable_code := 55, [86].LeakTest.Detailed.element_data[6].prec_code := 3, [86].LeakTest.Detailed.element_data[6].Unit_code := 12, [86].LeakTest.Detailed.element_data[6].result_measurement := 5.2330036, [86].LeakTest.Detailed.element_data[7].Variable_code := 58, [86].LeakTest.Detailed.element_data[7].prec_code := 2, [86].LeakTest.Detailed.element_data[7].Unit_code := 60, [86].LeakTest.Detailed.element_data[7].result_measurement := -1.0002404, [86].LeakTest.Detailed.element_data[8].Variable_code := 59, [86].LeakTest.Detailed.element_data[8].prec_code := 2, [86].LeakTest.Detailed.element_data[8].Unit_code := 60, [86].LeakTest.Detailed.element_data[8].result_measurement := 1.0002404, [86].LeakTest.Detailed.element_data[9].Variable_code := 12, [86].LeakTest.Detailed.element_data[9].prec_code := 3, [86].LeakTest.Detailed.element_data[9].Unit_code := 12, [86].LeakTest.Detailed.element_data[9].result_measurement := 5.000001, [86].LeakTest.Detailed.element_data[10].Variable_code := 62, [86].LeakTest.Detailed.element_data[10].prec_code := 2, [86].LeakTest.Detailed.element_data[10].Unit_code := 60, [86].LeakTest.Detailed.element_data[10].result_measurement := 1.1298805, [86].LeakTest.Detailed.element_data[11].Variable_code := 21, [86].LeakTest.Detailed.element_data[11].prec_code := 3, [86].LeakTest.Detailed.element_data[11].Unit_code := 41, [86].LeakTest.Detailed.element_data[11].result_measurement := 4.656613e-06, [86].LeakTest.Detailed.element_data[12].Variable_code := 25, [86].LeakTest.Detailed.element_data[12].prec_code := 3, [86].LeakTest.Detailed.element_data[12].Unit_code := 41, [86].LeakTest.Detailed.element_data[12].result_measurement := 0.023245811, [86].LeakTest.Detailed.element_data[13].Variable_code := 216, [86].LeakTest.Detailed.element_data[13].prec_code := 3, [86].LeakTest.Detailed.element_data[13].Unit_code := 41, [86].LeakTest.Detailed.element_data[13].result_measurement := -3.7252903e-05, [86].LeakTest.Detailed.element_data[14].Variable_code := 218, [86].LeakTest.Detailed.element_data[14].prec_code := 3, [86].LeakTest.Detailed.element_data[14].Unit_code := 41, [86].LeakTest.Detailed.element_data[14].result_measurement := 0.011632219, [86].LeakTest.Detailed.element_data[15].Variable_code := 295, [86].LeakTest.Detailed.element_data[15].prec_code := 3, [86].LeakTest.Detailed.element_data[15].Unit_code := 12, [86].LeakTest.Detailed.element_data[15].result_measurement := 5.2343307, [87].Barcode := 'B252620969', [87].VolumeTest.UID := 41955, [87].VolumeTest.Basic.unique_id := 41955, [87].VolumeTest.Basic.channel_num := 1, [87].VolumeTest.Basic.program_num := 1, [87].VolumeTest.Basic.evaluation_code := 1, [87].VolumeTest.Basic.test_port := 1, [87].VolumeTest.Basic.year := 26, [87].VolumeTest.Basic.month := 6, [87].VolumeTest.Basic.date := 4, [87].VolumeTest.Basic.hour := 14, [87].VolumeTest.Basic.minute := 58, [87].VolumeTest.Basic.second := 18, [87].VolumeTest.Basic.flags := 12, [87].VolumeTest.Basic.Num_tests := 1, [87].VolumeTest.Basic.test_elements.test_type := 69, [87].VolumeTest.Basic.test_elements.test_eval := 1, [87].VolumeTest.Basic.test_elements.num_elements := 4, [87].VolumeTest.Detailed.unique_id := 41955, [87].VolumeTest.Detailed.num_elements := 4,
        [87].VolumeTest.Detailed.Test_Type := 69, [87].VolumeTest.Detailed.element_data[0].Variable_code := 245, [87].VolumeTest.Detailed.element_data[0].prec_code := 2, [87].VolumeTest.Detailed.element_data[0].Unit_code := 165, [87].VolumeTest.Detailed.element_data[0].result_measurement := 186.52744, [87].VolumeTest.Detailed.element_data[1].Variable_code := 13, [87].VolumeTest.Detailed.element_data[1].prec_code := 3, [87].VolumeTest.Detailed.element_data[1].Unit_code := 12, [87].VolumeTest.Detailed.element_data[1].result_measurement := 1.782449, [87].VolumeTest.Detailed.element_data[2].Variable_code := 247, [87].VolumeTest.Detailed.element_data[2].prec_code := 3, [87].VolumeTest.Detailed.element_data[2].Unit_code := 12, [87].VolumeTest.Detailed.element_data[2].result_measurement := 5.1072054, [87].VolumeTest.Detailed.element_data[3].Variable_code := 295, [87].VolumeTest.Detailed.element_data[3].prec_code := 3, [87].VolumeTest.Detailed.element_data[3].Unit_code := 12, [87].VolumeTest.Detailed.element_data[3].result_measurement := 5.109105, [87].LeakTest.UID := 41956, [87].LeakTest.Basic.unique_id := 41956, [87].LeakTest.Basic.channel_num := 1, [87].LeakTest.Basic.program_num := 2, [87].LeakTest.Basic.evaluation_code := 1, [87].LeakTest.Basic.test_port := 1, [87].LeakTest.Basic.year := 26, [87].LeakTest.Basic.month := 6, [87].LeakTest.Basic.date := 4, [87].LeakTest.Basic.hour := 14, [87].LeakTest.Basic.minute := 58, [87].LeakTest.Basic.second := 25, [87].LeakTest.Basic.flags := 12, [87].LeakTest.Basic.Num_tests := 1, [87].LeakTest.Basic.test_elements.test_type := 66, [87].LeakTest.Basic.test_elements.test_eval := 1, [87].LeakTest.Basic.test_elements.num_elements := 16, [87].LeakTest.Detailed.unique_id := 41956, [87].LeakTest.Detailed.num_elements := 16, [87].LeakTest.Detailed.Test_Type := 66, [87].LeakTest.Detailed.element_data[0].Variable_code := 61, [87].LeakTest.Detailed.element_data[0].prec_code := 2, [87].LeakTest.Detailed.element_data[0].Unit_code := 60, [87].LeakTest.Detailed.element_data[0].result_measurement := -0.06984919, [87].LeakTest.Detailed.element_data[1].Variable_code := 28, [87].LeakTest.Detailed.element_data[1].prec_code := 3, [87].LeakTest.Detailed.element_data[1].Unit_code := 41, [87].LeakTest.Detailed.element_data[1].result_measurement := 0.00022817403, [87].LeakTest.Detailed.element_data[2].Variable_code := 13, [87].LeakTest.Detailed.element_data[2].prec_code := 3, [87].LeakTest.Detailed.element_data[2].Unit_code := 12, [87].LeakTest.Detailed.element_data[2].result_measurement := 5.137343, [87].LeakTest.Detailed.element_data[3].Variable_code := 75, [87].LeakTest.Detailed.element_data[3].prec_code := 2, [87].LeakTest.Detailed.element_data[3].Unit_code := 60, [87].LeakTest.Detailed.element_data[4].Variable_code := 60, [87].LeakTest.Detailed.element_data[4].prec_code := 2, [87].LeakTest.Detailed.element_data[4].Unit_code := 60, [87].LeakTest.Detailed.element_data[4].result_measurement := -0.07878989, [87].LeakTest.Detailed.element_data[5].Variable_code := 56, [87].LeakTest.Detailed.element_data[5].prec_code := 3, [87].LeakTest.Detailed.element_data[5].Unit_code := 41, [87].LeakTest.Detailed.element_data[5].result_measurement := 0.00013038516,
        [87].LeakTest.Detailed.element_data[6].Variable_code := 55, [87].LeakTest.Detailed.element_data[6].prec_code := 3, [87].LeakTest.Detailed.element_data[6].Unit_code := 12, [87].LeakTest.Detailed.element_data[6].result_measurement := 5.137343, [87].LeakTest.Detailed.element_data[7].Variable_code := 58, [87].LeakTest.Detailed.element_data[7].prec_code := 2, [87].LeakTest.Detailed.element_data[7].Unit_code := 60, [87].LeakTest.Detailed.element_data[7].result_measurement := -1.0002404, [87].LeakTest.Detailed.element_data[8].Variable_code := 59, [87].LeakTest.Detailed.element_data[8].prec_code := 2, [87].LeakTest.Detailed.element_data[8].Unit_code := 60, [87].LeakTest.Detailed.element_data[8].result_measurement := 1.0002404, [87].LeakTest.Detailed.element_data[9].Variable_code := 12, [87].LeakTest.Detailed.element_data[9].prec_code := 3, [87].LeakTest.Detailed.element_data[9].Unit_code := 12, [87].LeakTest.Detailed.element_data[9].result_measurement := 5.000001, [87].LeakTest.Detailed.element_data[10].Variable_code := 62, [87].LeakTest.Detailed.element_data[10].prec_code := 2, [87].LeakTest.Detailed.element_data[10].Unit_code := 60, [87].LeakTest.Detailed.element_data[10].result_measurement := 1.1002644, [87].LeakTest.Detailed.element_data[11].Variable_code := 21, [87].LeakTest.Detailed.element_data[11].prec_code := 3, [87].LeakTest.Detailed.element_data[11].Unit_code := 41, [87].LeakTest.Detailed.element_data[11].result_measurement := 0.0015180558, [87].LeakTest.Detailed.element_data[12].Variable_code := 25, [87].LeakTest.Detailed.element_data[12].prec_code := 3, [87].LeakTest.Detailed.element_data[12].Unit_code := 41, [87].LeakTest.Detailed.element_data[12].result_measurement := 0.021727756, [87].LeakTest.Detailed.element_data[13].Variable_code := 216, [87].LeakTest.Detailed.element_data[13].prec_code := 3, [87].LeakTest.Detailed.element_data[13].Unit_code := 41, [87].LeakTest.Detailed.element_data[13].result_measurement := 0.00085681677, [87].LeakTest.Detailed.element_data[14].Variable_code := 218, [87].LeakTest.Detailed.element_data[14].prec_code := 3, [87].LeakTest.Detailed.element_data[14].Unit_code := 41, [87].LeakTest.Detailed.element_data[14].result_measurement := 0.01094304, [87].LeakTest.Detailed.element_data[15].Variable_code := 295, [87].LeakTest.Detailed.element_data[15].prec_code := 3, [87].LeakTest.Detailed.element_data[15].Unit_code := 12, [87].LeakTest.Detailed.element_data[15].result_measurement := 5.1386003, [88].Barcode := 'B252620970', [88].VolumeTest.UID := 42949, [88].VolumeTest.Basic.unique_id := 42949, [88].VolumeTest.Basic.channel_num := 1, [88].VolumeTest.Basic.program_num := 1, [88].VolumeTest.Basic.evaluation_code := 1, [88].VolumeTest.Basic.test_port := 1, [88].VolumeTest.Basic.year := 26, [88].VolumeTest.Basic.month := 6, [88].VolumeTest.Basic.date := 4, [88].VolumeTest.Basic.hour := 14, [88].VolumeTest.Basic.minute := 59, [88].VolumeTest.Basic.second := 45, [88].VolumeTest.Basic.flags := 12, [88].VolumeTest.Basic.Num_tests := 1, [88].VolumeTest.Basic.test_elements.test_type := 69, [88].VolumeTest.Basic.test_elements.test_eval := 1, [88].VolumeTest.Basic.test_elements.num_elements := 4, [88].VolumeTest.Detailed.unique_id := 42949, [88].VolumeTest.Detailed.num_elements := 4,
        [88].VolumeTest.Detailed.Test_Type := 69, [88].VolumeTest.Detailed.element_data[0].Variable_code := 245, [88].VolumeTest.Detailed.element_data[0].prec_code := 2, [88].VolumeTest.Detailed.element_data[0].Unit_code := 165, [88].VolumeTest.Detailed.element_data[0].result_measurement := 188.34744, [88].VolumeTest.Detailed.element_data[1].Variable_code := 13, [88].VolumeTest.Detailed.element_data[1].prec_code := 3, [88].VolumeTest.Detailed.element_data[1].Unit_code := 12, [88].VolumeTest.Detailed.element_data[1].result_measurement := 1.8081255, [88].VolumeTest.Detailed.element_data[2].Variable_code := 247, [88].VolumeTest.Detailed.element_data[2].prec_code := 3, [88].VolumeTest.Detailed.element_data[2].Unit_code := 12, [88].VolumeTest.Detailed.element_data[2].result_measurement := 5.2136836, [88].VolumeTest.Detailed.element_data[3].Variable_code := 295, [88].VolumeTest.Detailed.element_data[3].prec_code := 3, [88].VolumeTest.Detailed.element_data[3].Unit_code := 12, [88].VolumeTest.Detailed.element_data[3].result_measurement := 5.2160025, [88].LeakTest.UID := 42950, [88].LeakTest.Basic.unique_id := 42950, [88].LeakTest.Basic.channel_num := 1, [88].LeakTest.Basic.program_num := 2, [88].LeakTest.Basic.evaluation_code := 1, [88].LeakTest.Basic.test_port := 1, [88].LeakTest.Basic.year := 26, [88].LeakTest.Basic.month := 6, [88].LeakTest.Basic.date := 4, [88].LeakTest.Basic.hour := 14, [88].LeakTest.Basic.minute := 59, [88].LeakTest.Basic.second := 52, [88].LeakTest.Basic.flags := 12, [88].LeakTest.Basic.Num_tests := 1, [88].LeakTest.Basic.test_elements.test_type := 66, [88].LeakTest.Basic.test_elements.test_eval := 1, [88].LeakTest.Basic.test_elements.num_elements := 16, [88].LeakTest.Detailed.unique_id := 42950, [88].LeakTest.Detailed.num_elements := 16, [88].LeakTest.Detailed.Test_Type := 66, [88].LeakTest.Detailed.element_data[0].Variable_code := 61, [88].LeakTest.Detailed.element_data[0].prec_code := 2, [88].LeakTest.Detailed.element_data[0].Unit_code := 60, [88].LeakTest.Detailed.element_data[0].result_measurement := -0.003911555, [88].LeakTest.Detailed.element_data[1].Variable_code := 28, [88].LeakTest.Detailed.element_data[1].prec_code := 3, [88].LeakTest.Detailed.element_data[1].Unit_code := 41, [88].LeakTest.Detailed.element_data[1].result_measurement := -7.916242e-05, [88].LeakTest.Detailed.element_data[2].Variable_code := 13, [88].LeakTest.Detailed.element_data[2].prec_code := 3, [88].LeakTest.Detailed.element_data[2].Unit_code := 12, [88].LeakTest.Detailed.element_data[2].result_measurement := 5.2312574, [88].LeakTest.Detailed.element_data[3].Variable_code := 75, [88].LeakTest.Detailed.element_data[3].prec_code := 2, [88].LeakTest.Detailed.element_data[3].Unit_code := 60, [88].LeakTest.Detailed.element_data[4].Variable_code := 60, [88].LeakTest.Detailed.element_data[4].prec_code := 2, [88].LeakTest.Detailed.element_data[4].Unit_code := 60, [88].LeakTest.Detailed.element_data[4].result_measurement := -0.012293458, [88].LeakTest.Detailed.element_data[5].Variable_code := 56, [88].LeakTest.Detailed.element_data[5].prec_code := 3, [88].LeakTest.Detailed.element_data[5].Unit_code := 41, [88].LeakTest.Detailed.element_data[5].result_measurement := -0.00016763806,
        [88].LeakTest.Detailed.element_data[6].Variable_code := 55, [88].LeakTest.Detailed.element_data[6].prec_code := 3, [88].LeakTest.Detailed.element_data[6].Unit_code := 12, [88].LeakTest.Detailed.element_data[6].result_measurement := 5.2312574, [88].LeakTest.Detailed.element_data[7].Variable_code := 58, [88].LeakTest.Detailed.element_data[7].prec_code := 2, [88].LeakTest.Detailed.element_data[7].Unit_code := 60, [88].LeakTest.Detailed.element_data[7].result_measurement := -1.0002404, [88].LeakTest.Detailed.element_data[8].Variable_code := 59, [88].LeakTest.Detailed.element_data[8].prec_code := 2, [88].LeakTest.Detailed.element_data[8].Unit_code := 60, [88].LeakTest.Detailed.element_data[8].result_measurement := 1.0002404, [88].LeakTest.Detailed.element_data[9].Variable_code := 12, [88].LeakTest.Detailed.element_data[9].prec_code := 3, [88].LeakTest.Detailed.element_data[9].Unit_code := 12, [88].LeakTest.Detailed.element_data[9].result_measurement := 5.000001, [88].LeakTest.Detailed.element_data[10].Variable_code := 62, [88].LeakTest.Detailed.element_data[10].prec_code := 2, [88].LeakTest.Detailed.element_data[10].Unit_code := 60, [88].LeakTest.Detailed.element_data[10].result_measurement := 1.1298805, [88].LeakTest.Detailed.element_data[11].Variable_code := 21, [88].LeakTest.Detailed.element_data[11].prec_code := 3, [88].LeakTest.Detailed.element_data[11].Unit_code := 41, [88].LeakTest.Detailed.element_data[11].result_measurement := 4.656613e-06, [88].LeakTest.Detailed.element_data[12].Variable_code := 25, [88].LeakTest.Detailed.element_data[12].prec_code := 3, [88].LeakTest.Detailed.element_data[12].Unit_code := 41, [88].LeakTest.Detailed.element_data[12].result_measurement := 0.023245811, [88].LeakTest.Detailed.element_data[13].Variable_code := 216, [88].LeakTest.Detailed.element_data[13].prec_code := 3, [88].LeakTest.Detailed.element_data[13].Unit_code := 41, [88].LeakTest.Detailed.element_data[13].result_measurement := -3.7252903e-05, [88].LeakTest.Detailed.element_data[14].Variable_code := 218, [88].LeakTest.Detailed.element_data[14].prec_code := 3, [88].LeakTest.Detailed.element_data[14].Unit_code := 41, [88].LeakTest.Detailed.element_data[14].result_measurement := 0.011632219, [88].LeakTest.Detailed.element_data[15].Variable_code := 295, [88].LeakTest.Detailed.element_data[15].prec_code := 3, [88].LeakTest.Detailed.element_data[15].Unit_code := 12, [88].LeakTest.Detailed.element_data[15].result_measurement := 5.2330365, [89].Barcode := 'B252620863', [89].VolumeTest.UID := 42952, [89].VolumeTest.Basic.unique_id := 42952, [89].VolumeTest.Basic.channel_num := 1, [89].VolumeTest.Basic.program_num := 1, [89].VolumeTest.Basic.evaluation_code := 1, [89].VolumeTest.Basic.test_port := 1, [89].VolumeTest.Basic.year := 26, [89].VolumeTest.Basic.month := 6, [89].VolumeTest.Basic.date := 4, [89].VolumeTest.Basic.hour := 15, [89].VolumeTest.Basic.minute := 3, [89].VolumeTest.Basic.second := 30, [89].VolumeTest.Basic.flags := 12, [89].VolumeTest.Basic.Num_tests := 1, [89].VolumeTest.Basic.test_elements.test_type := 69, [89].VolumeTest.Basic.test_elements.test_eval := 1, [89].VolumeTest.Basic.test_elements.num_elements := 4, [89].VolumeTest.Detailed.unique_id := 42952, [89].VolumeTest.Detailed.num_elements := 4,
        [89].VolumeTest.Detailed.Test_Type := 69, [89].VolumeTest.Detailed.element_data[0].Variable_code := 245, [89].VolumeTest.Detailed.element_data[0].prec_code := 2, [89].VolumeTest.Detailed.element_data[0].Unit_code := 165, [89].VolumeTest.Detailed.element_data[0].result_measurement := 188.1703, [89].VolumeTest.Detailed.element_data[1].Variable_code := 13, [89].VolumeTest.Detailed.element_data[1].prec_code := 3, [89].VolumeTest.Detailed.element_data[1].Unit_code := 12, [89].VolumeTest.Detailed.element_data[1].result_measurement := 1.8089218, [89].VolumeTest.Detailed.element_data[2].Variable_code := 247, [89].VolumeTest.Detailed.element_data[2].prec_code := 3, [89].VolumeTest.Detailed.element_data[2].Unit_code := 12, [89].VolumeTest.Detailed.element_data[2].result_measurement := 5.212775, [89].VolumeTest.Detailed.element_data[3].Variable_code := 295, [89].VolumeTest.Detailed.element_data[3].prec_code := 3, [89].VolumeTest.Detailed.element_data[3].Unit_code := 12, [89].VolumeTest.Detailed.element_data[3].result_measurement := 5.214061, [89].LeakTest.UID := 42953, [89].LeakTest.Basic.unique_id := 42953, [89].LeakTest.Basic.channel_num := 1, [89].LeakTest.Basic.program_num := 2, [89].LeakTest.Basic.evaluation_code := 1, [89].LeakTest.Basic.test_port := 1, [89].LeakTest.Basic.year := 26, [89].LeakTest.Basic.month := 6, [89].LeakTest.Basic.date := 4, [89].LeakTest.Basic.hour := 15, [89].LeakTest.Basic.minute := 3, [89].LeakTest.Basic.second := 37, [89].LeakTest.Basic.flags := 12, [89].LeakTest.Basic.Num_tests := 1, [89].LeakTest.Basic.test_elements.test_type := 66, [89].LeakTest.Basic.test_elements.test_eval := 1, [89].LeakTest.Basic.test_elements.num_elements := 16, [89].LeakTest.Detailed.unique_id := 42953, [89].LeakTest.Detailed.num_elements := 16, [89].LeakTest.Detailed.Test_Type := 66, [89].LeakTest.Detailed.element_data[0].Variable_code := 61, [89].LeakTest.Detailed.element_data[0].prec_code := 2, [89].LeakTest.Detailed.element_data[0].Unit_code := 60, [89].LeakTest.Detailed.element_data[0].result_measurement := 0.0055879354, [89].LeakTest.Detailed.element_data[1].Variable_code := 28, [89].LeakTest.Detailed.element_data[1].prec_code := 3, [89].LeakTest.Detailed.element_data[1].Unit_code := 41, [89].LeakTest.Detailed.element_data[1].result_measurement := 0.00012572855, [89].LeakTest.Detailed.element_data[2].Variable_code := 13, [89].LeakTest.Detailed.element_data[2].prec_code := 3, [89].LeakTest.Detailed.element_data[2].Unit_code := 12, [89].LeakTest.Detailed.element_data[2].result_measurement := 5.2312155, [89].LeakTest.Detailed.element_data[3].Variable_code := 75, [89].LeakTest.Detailed.element_data[3].prec_code := 2, [89].LeakTest.Detailed.element_data[3].Unit_code := 60, [89].LeakTest.Detailed.element_data[4].Variable_code := 60, [89].LeakTest.Detailed.element_data[4].prec_code := 2, [89].LeakTest.Detailed.element_data[4].Unit_code := 60, [89].LeakTest.Detailed.element_data[4].result_measurement := 0.0044703484, [89].LeakTest.Detailed.element_data[5].Variable_code := 56, [89].LeakTest.Detailed.element_data[5].prec_code := 3, [89].LeakTest.Detailed.element_data[5].Unit_code := 41, [89].LeakTest.Detailed.element_data[5].result_measurement := 1.3969839e-05,
        [89].LeakTest.Detailed.element_data[6].Variable_code := 55, [89].LeakTest.Detailed.element_data[6].prec_code := 3, [89].LeakTest.Detailed.element_data[6].Unit_code := 12, [89].LeakTest.Detailed.element_data[6].result_measurement := 5.2312155, [89].LeakTest.Detailed.element_data[7].Variable_code := 58, [89].LeakTest.Detailed.element_data[7].prec_code := 2, [89].LeakTest.Detailed.element_data[7].Unit_code := 60, [89].LeakTest.Detailed.element_data[7].result_measurement := -1.0002404, [89].LeakTest.Detailed.element_data[8].Variable_code := 59, [89].LeakTest.Detailed.element_data[8].prec_code := 2, [89].LeakTest.Detailed.element_data[8].Unit_code := 60, [89].LeakTest.Detailed.element_data[8].result_measurement := 1.0002404, [89].LeakTest.Detailed.element_data[9].Variable_code := 12, [89].LeakTest.Detailed.element_data[9].prec_code := 3, [89].LeakTest.Detailed.element_data[9].Unit_code := 12, [89].LeakTest.Detailed.element_data[9].result_measurement := 5.000001, [89].LeakTest.Detailed.element_data[10].Variable_code := 62, [89].LeakTest.Detailed.element_data[10].prec_code := 2, [89].LeakTest.Detailed.element_data[10].Unit_code := 60, [89].LeakTest.Detailed.element_data[10].result_measurement := 1.1298805, [89].LeakTest.Detailed.element_data[11].Variable_code := 21, [89].LeakTest.Detailed.element_data[11].prec_code := 3, [89].LeakTest.Detailed.element_data[11].Unit_code := 41, [89].LeakTest.Detailed.element_data[11].result_measurement := 4.656613e-06, [89].LeakTest.Detailed.element_data[12].Variable_code := 25, [89].LeakTest.Detailed.element_data[12].prec_code := 3, [89].LeakTest.Detailed.element_data[12].Unit_code := 41, [89].LeakTest.Detailed.element_data[12].result_measurement := 0.023245811, [89].LeakTest.Detailed.element_data[13].Variable_code := 216, [89].LeakTest.Detailed.element_data[13].prec_code := 3, [89].LeakTest.Detailed.element_data[13].Unit_code := 41, [89].LeakTest.Detailed.element_data[13].result_measurement := -3.7252903e-05, [89].LeakTest.Detailed.element_data[14].Variable_code := 218, [89].LeakTest.Detailed.element_data[14].prec_code := 3, [89].LeakTest.Detailed.element_data[14].Unit_code := 41, [89].LeakTest.Detailed.element_data[14].result_measurement := 0.011632219, [89].LeakTest.Detailed.element_data[15].Variable_code := 295, [89].LeakTest.Detailed.element_data[15].prec_code := 3, [89].LeakTest.Detailed.element_data[15].Unit_code := 12, [89].LeakTest.Detailed.element_data[15].result_measurement := 5.2327847, [90].Barcode := 'B252620969', [90].VolumeTest.UID := 41958, [90].VolumeTest.Basic.unique_id := 41958, [90].VolumeTest.Basic.channel_num := 1, [90].VolumeTest.Basic.program_num := 1, [90].VolumeTest.Basic.evaluation_code := 1, [90].VolumeTest.Basic.test_port := 1, [90].VolumeTest.Basic.year := 26, [90].VolumeTest.Basic.month := 6, [90].VolumeTest.Basic.date := 4, [90].VolumeTest.Basic.hour := 15, [90].VolumeTest.Basic.minute := 3, [90].VolumeTest.Basic.second := 10, [90].VolumeTest.Basic.flags := 12, [90].VolumeTest.Basic.Num_tests := 1, [90].VolumeTest.Basic.test_elements.test_type := 69, [90].VolumeTest.Basic.test_elements.test_eval := 1, [90].VolumeTest.Basic.test_elements.num_elements := 4, [90].VolumeTest.Detailed.unique_id := 41958, [90].VolumeTest.Detailed.num_elements := 4,
        [90].VolumeTest.Detailed.Test_Type := 69, [90].VolumeTest.Detailed.element_data[0].Variable_code := 245, [90].VolumeTest.Detailed.element_data[0].prec_code := 2, [90].VolumeTest.Detailed.element_data[0].Unit_code := 165, [90].VolumeTest.Detailed.element_data[0].result_measurement := 186.90665, [90].VolumeTest.Detailed.element_data[1].Variable_code := 13, [90].VolumeTest.Detailed.element_data[1].prec_code := 3, [90].VolumeTest.Detailed.element_data[1].Unit_code := 12, [90].VolumeTest.Detailed.element_data[1].result_measurement := 1.7801206, [90].VolumeTest.Detailed.element_data[2].Variable_code := 247, [90].VolumeTest.Detailed.element_data[2].prec_code := 3, [90].VolumeTest.Detailed.element_data[2].Unit_code := 12, [90].VolumeTest.Detailed.element_data[2].result_measurement := 5.1072845, [90].VolumeTest.Detailed.element_data[3].Variable_code := 295, [90].VolumeTest.Detailed.element_data[3].prec_code := 3, [90].VolumeTest.Detailed.element_data[3].Unit_code := 12, [90].VolumeTest.Detailed.element_data[3].result_measurement := 5.1086583, [90].LeakTest.UID := 41959, [90].LeakTest.Basic.unique_id := 41959, [90].LeakTest.Basic.channel_num := 1, [90].LeakTest.Basic.program_num := 2, [90].LeakTest.Basic.evaluation_code := 1, [90].LeakTest.Basic.test_port := 1, [90].LeakTest.Basic.year := 26, [90].LeakTest.Basic.month := 6, [90].LeakTest.Basic.date := 4, [90].LeakTest.Basic.hour := 15, [90].LeakTest.Basic.minute := 3, [90].LeakTest.Basic.second := 17, [90].LeakTest.Basic.flags := 12, [90].LeakTest.Basic.Num_tests := 1, [90].LeakTest.Basic.test_elements.test_type := 66, [90].LeakTest.Basic.test_elements.test_eval := 1, [90].LeakTest.Basic.test_elements.num_elements := 16, [90].LeakTest.Detailed.unique_id := 41959, [90].LeakTest.Detailed.num_elements := 16, [90].LeakTest.Detailed.Test_Type := 66, [90].LeakTest.Detailed.element_data[0].Variable_code := 61, [90].LeakTest.Detailed.element_data[0].prec_code := 2, [90].LeakTest.Detailed.element_data[0].Unit_code := 60, [90].LeakTest.Detailed.element_data[0].result_measurement := -0.06258488, [90].LeakTest.Detailed.element_data[1].Variable_code := 28, [90].LeakTest.Detailed.element_data[1].prec_code := 3, [90].LeakTest.Detailed.element_data[1].Unit_code := 41, [90].LeakTest.Detailed.element_data[1].result_measurement := 0.00036787242, [90].LeakTest.Detailed.element_data[2].Variable_code := 13, [90].LeakTest.Detailed.element_data[2].prec_code := 3, [90].LeakTest.Detailed.element_data[2].Unit_code := 12, [90].LeakTest.Detailed.element_data[2].result_measurement := 5.1356993, [90].LeakTest.Detailed.element_data[3].Variable_code := 75, [90].LeakTest.Detailed.element_data[3].prec_code := 2, [90].LeakTest.Detailed.element_data[3].Unit_code := 60, [90].LeakTest.Detailed.element_data[4].Variable_code := 60, [90].LeakTest.Detailed.element_data[4].prec_code := 2, [90].LeakTest.Detailed.element_data[4].Unit_code := 60, [90].LeakTest.Detailed.element_data[4].result_measurement := -0.073201954, [90].LeakTest.Detailed.element_data[5].Variable_code := 56, [90].LeakTest.Detailed.element_data[5].prec_code := 3, [90].LeakTest.Detailed.element_data[5].Unit_code := 41, [90].LeakTest.Detailed.element_data[5].result_measurement := 0.0001816079,
        [90].LeakTest.Detailed.element_data[6].Variable_code := 55, [90].LeakTest.Detailed.element_data[6].prec_code := 3, [90].LeakTest.Detailed.element_data[6].Unit_code := 12, [90].LeakTest.Detailed.element_data[6].result_measurement := 5.1356993, [90].LeakTest.Detailed.element_data[7].Variable_code := 58, [90].LeakTest.Detailed.element_data[7].prec_code := 2, [90].LeakTest.Detailed.element_data[7].Unit_code := 60, [90].LeakTest.Detailed.element_data[7].result_measurement := -1.0002404, [90].LeakTest.Detailed.element_data[8].Variable_code := 59, [90].LeakTest.Detailed.element_data[8].prec_code := 2, [90].LeakTest.Detailed.element_data[8].Unit_code := 60, [90].LeakTest.Detailed.element_data[8].result_measurement := 1.0002404, [90].LeakTest.Detailed.element_data[9].Variable_code := 12, [90].LeakTest.Detailed.element_data[9].prec_code := 3, [90].LeakTest.Detailed.element_data[9].Unit_code := 12, [90].LeakTest.Detailed.element_data[9].result_measurement := 5.000001, [90].LeakTest.Detailed.element_data[10].Variable_code := 62, [90].LeakTest.Detailed.element_data[10].prec_code := 2, [90].LeakTest.Detailed.element_data[10].Unit_code := 60, [90].LeakTest.Detailed.element_data[10].result_measurement := 1.1002644, [90].LeakTest.Detailed.element_data[11].Variable_code := 21, [90].LeakTest.Detailed.element_data[11].prec_code := 3, [90].LeakTest.Detailed.element_data[11].Unit_code := 41, [90].LeakTest.Detailed.element_data[11].result_measurement := 0.0015180558, [90].LeakTest.Detailed.element_data[12].Variable_code := 25, [90].LeakTest.Detailed.element_data[12].prec_code := 3, [90].LeakTest.Detailed.element_data[12].Unit_code := 41, [90].LeakTest.Detailed.element_data[12].result_measurement := 0.021727756, [90].LeakTest.Detailed.element_data[13].Variable_code := 216, [90].LeakTest.Detailed.element_data[13].prec_code := 3, [90].LeakTest.Detailed.element_data[13].Unit_code := 41, [90].LeakTest.Detailed.element_data[13].result_measurement := 0.00085681677, [90].LeakTest.Detailed.element_data[14].Variable_code := 218, [90].LeakTest.Detailed.element_data[14].prec_code := 3, [90].LeakTest.Detailed.element_data[14].Unit_code := 41, [90].LeakTest.Detailed.element_data[14].result_measurement := 0.01094304, [90].LeakTest.Detailed.element_data[15].Variable_code := 295, [90].LeakTest.Detailed.element_data[15].prec_code := 3, [90].LeakTest.Detailed.element_data[15].Unit_code := 12, [90].LeakTest.Detailed.element_data[15].result_measurement := 5.1374407, [91].Barcode := 'B252620969', [91].VolumeTest.UID := 41961, [91].VolumeTest.Basic.unique_id := 41961, [91].VolumeTest.Basic.channel_num := 1, [91].VolumeTest.Basic.program_num := 1, [91].VolumeTest.Basic.evaluation_code := 1, [91].VolumeTest.Basic.test_port := 1, [91].VolumeTest.Basic.year := 26, [91].VolumeTest.Basic.month := 6, [91].VolumeTest.Basic.date := 4, [91].VolumeTest.Basic.hour := 15, [91].VolumeTest.Basic.minute := 6, [91].VolumeTest.Basic.second := 33, [91].VolumeTest.Basic.flags := 12, [91].VolumeTest.Basic.Num_tests := 1, [91].VolumeTest.Basic.test_elements.test_type := 69, [91].VolumeTest.Basic.test_elements.test_eval := 1, [91].VolumeTest.Basic.test_elements.num_elements := 4, [91].VolumeTest.Detailed.unique_id := 41961, [91].VolumeTest.Detailed.num_elements := 4,
        [91].VolumeTest.Detailed.Test_Type := 69, [91].VolumeTest.Detailed.element_data[0].Variable_code := 245, [91].VolumeTest.Detailed.element_data[0].prec_code := 2, [91].VolumeTest.Detailed.element_data[0].Unit_code := 165, [91].VolumeTest.Detailed.element_data[0].result_measurement := 186.6259, [91].VolumeTest.Detailed.element_data[1].Variable_code := 13, [91].VolumeTest.Detailed.element_data[1].prec_code := 3, [91].VolumeTest.Detailed.element_data[1].Unit_code := 12, [91].VolumeTest.Detailed.element_data[1].result_measurement := 1.7820624, [91].VolumeTest.Detailed.element_data[2].Variable_code := 247, [91].VolumeTest.Detailed.element_data[2].prec_code := 3, [91].VolumeTest.Detailed.element_data[2].Unit_code := 12, [91].VolumeTest.Detailed.element_data[2].result_measurement := 5.1078525, [91].VolumeTest.Detailed.element_data[3].Variable_code := 295, [91].VolumeTest.Detailed.element_data[3].prec_code := 3, [91].VolumeTest.Detailed.element_data[3].Unit_code := 12, [91].VolumeTest.Detailed.element_data[3].result_measurement := 5.1083417, [91].LeakTest.UID := 41962, [91].LeakTest.Basic.unique_id := 41962, [91].LeakTest.Basic.channel_num := 1, [91].LeakTest.Basic.program_num := 2, [91].LeakTest.Basic.evaluation_code := 1, [91].LeakTest.Basic.test_port := 1, [91].LeakTest.Basic.year := 26, [91].LeakTest.Basic.month := 6, [91].LeakTest.Basic.date := 4, [91].LeakTest.Basic.hour := 15, [91].LeakTest.Basic.minute := 6, [91].LeakTest.Basic.second := 39, [91].LeakTest.Basic.flags := 12, [91].LeakTest.Basic.Num_tests := 1, [91].LeakTest.Basic.test_elements.test_type := 66, [91].LeakTest.Basic.test_elements.test_eval := 1, [91].LeakTest.Basic.test_elements.num_elements := 16, [91].LeakTest.Detailed.unique_id := 41962, [91].LeakTest.Detailed.num_elements := 16, [91].LeakTest.Detailed.Test_Type := 66, [91].LeakTest.Detailed.element_data[0].Variable_code := 61, [91].LeakTest.Detailed.element_data[0].prec_code := 2, [91].LeakTest.Detailed.element_data[0].Unit_code := 60, [91].LeakTest.Detailed.element_data[0].result_measurement := -0.058673322, [91].LeakTest.Detailed.element_data[1].Variable_code := 28, [91].LeakTest.Detailed.element_data[1].prec_code := 3, [91].LeakTest.Detailed.element_data[1].Unit_code := 41, [91].LeakTest.Detailed.element_data[1].result_measurement := 0.000433065, [91].LeakTest.Detailed.element_data[2].Variable_code := 13, [91].LeakTest.Detailed.element_data[2].prec_code := 3, [91].LeakTest.Detailed.element_data[2].Unit_code := 12, [91].LeakTest.Detailed.element_data[2].result_measurement := 5.136598, [91].LeakTest.Detailed.element_data[3].Variable_code := 75, [91].LeakTest.Detailed.element_data[3].prec_code := 2, [91].LeakTest.Detailed.element_data[3].Unit_code := 60, [91].LeakTest.Detailed.element_data[4].Variable_code := 60, [91].LeakTest.Detailed.element_data[4].prec_code := 2, [91].LeakTest.Detailed.element_data[4].Unit_code := 60, [91].LeakTest.Detailed.element_data[4].result_measurement := -0.06649643, [91].LeakTest.Detailed.element_data[5].Variable_code := 56, [91].LeakTest.Detailed.element_data[5].prec_code := 3, [91].LeakTest.Detailed.element_data[5].Unit_code := 41, [91].LeakTest.Detailed.element_data[5].result_measurement := 0.00024214387,
        [91].LeakTest.Detailed.element_data[6].Variable_code := 55, [91].LeakTest.Detailed.element_data[6].prec_code := 3, [91].LeakTest.Detailed.element_data[6].Unit_code := 12, [91].LeakTest.Detailed.element_data[6].result_measurement := 5.136598, [91].LeakTest.Detailed.element_data[7].Variable_code := 58, [91].LeakTest.Detailed.element_data[7].prec_code := 2, [91].LeakTest.Detailed.element_data[7].Unit_code := 60, [91].LeakTest.Detailed.element_data[7].result_measurement := -1.0002404, [91].LeakTest.Detailed.element_data[8].Variable_code := 59, [91].LeakTest.Detailed.element_data[8].prec_code := 2, [91].LeakTest.Detailed.element_data[8].Unit_code := 60, [91].LeakTest.Detailed.element_data[8].result_measurement := 1.0002404, [91].LeakTest.Detailed.element_data[9].Variable_code := 12, [91].LeakTest.Detailed.element_data[9].prec_code := 3, [91].LeakTest.Detailed.element_data[9].Unit_code := 12, [91].LeakTest.Detailed.element_data[9].result_measurement := 5.000001, [91].LeakTest.Detailed.element_data[10].Variable_code := 62, [91].LeakTest.Detailed.element_data[10].prec_code := 2, [91].LeakTest.Detailed.element_data[10].Unit_code := 60, [91].LeakTest.Detailed.element_data[10].result_measurement := 1.1002644, [91].LeakTest.Detailed.element_data[11].Variable_code := 21, [91].LeakTest.Detailed.element_data[11].prec_code := 3, [91].LeakTest.Detailed.element_data[11].Unit_code := 41, [91].LeakTest.Detailed.element_data[11].result_measurement := 0.0015180558, [91].LeakTest.Detailed.element_data[12].Variable_code := 25, [91].LeakTest.Detailed.element_data[12].prec_code := 3, [91].LeakTest.Detailed.element_data[12].Unit_code := 41, [91].LeakTest.Detailed.element_data[12].result_measurement := 0.021727756, [91].LeakTest.Detailed.element_data[13].Variable_code := 216, [91].LeakTest.Detailed.element_data[13].prec_code := 3, [91].LeakTest.Detailed.element_data[13].Unit_code := 41, [91].LeakTest.Detailed.element_data[13].result_measurement := 0.00085681677, [91].LeakTest.Detailed.element_data[14].Variable_code := 218, [91].LeakTest.Detailed.element_data[14].prec_code := 3, [91].LeakTest.Detailed.element_data[14].Unit_code := 41, [91].LeakTest.Detailed.element_data[14].result_measurement := 0.01094304, [91].LeakTest.Detailed.element_data[15].Variable_code := 295, [91].LeakTest.Detailed.element_data[15].prec_code := 3, [91].LeakTest.Detailed.element_data[15].Unit_code := 12, [91].LeakTest.Detailed.element_data[15].result_measurement := 5.1383443, [92].Barcode := 'B252620863', [92].VolumeTest.UID := 42955, [92].VolumeTest.Basic.unique_id := 42955, [92].VolumeTest.Basic.channel_num := 1, [92].VolumeTest.Basic.program_num := 1, [92].VolumeTest.Basic.evaluation_code := 1, [92].VolumeTest.Basic.test_port := 1, [92].VolumeTest.Basic.year := 26, [92].VolumeTest.Basic.month := 6, [92].VolumeTest.Basic.date := 4, [92].VolumeTest.Basic.hour := 15, [92].VolumeTest.Basic.minute := 6, [92].VolumeTest.Basic.second := 56, [92].VolumeTest.Basic.flags := 12, [92].VolumeTest.Basic.Num_tests := 1, [92].VolumeTest.Basic.test_elements.test_type := 69, [92].VolumeTest.Basic.test_elements.test_eval := 1, [92].VolumeTest.Basic.test_elements.num_elements := 4, [92].VolumeTest.Detailed.unique_id := 42955, [92].VolumeTest.Detailed.num_elements := 4,
        [92].VolumeTest.Detailed.Test_Type := 69, [92].VolumeTest.Detailed.element_data[0].Variable_code := 245, [92].VolumeTest.Detailed.element_data[0].prec_code := 2, [92].VolumeTest.Detailed.element_data[0].Unit_code := 165, [92].VolumeTest.Detailed.element_data[0].result_measurement := 188.15602, [92].VolumeTest.Detailed.element_data[1].Variable_code := 13, [92].VolumeTest.Detailed.element_data[1].prec_code := 3, [92].VolumeTest.Detailed.element_data[1].Unit_code := 12, [92].VolumeTest.Detailed.element_data[1].result_measurement := 1.809257, [92].VolumeTest.Detailed.element_data[2].Variable_code := 247, [92].VolumeTest.Detailed.element_data[2].prec_code := 3, [92].VolumeTest.Detailed.element_data[2].Unit_code := 12, [92].VolumeTest.Detailed.element_data[2].result_measurement := 5.2134833, [92].VolumeTest.Detailed.element_data[3].Variable_code := 295, [92].VolumeTest.Detailed.element_data[3].prec_code := 3, [92].VolumeTest.Detailed.element_data[3].Unit_code := 12, [92].VolumeTest.Detailed.element_data[3].result_measurement := 5.215304, [92].LeakTest.UID := 42956, [92].LeakTest.Basic.unique_id := 42956, [92].LeakTest.Basic.channel_num := 1, [92].LeakTest.Basic.program_num := 2, [92].LeakTest.Basic.evaluation_code := 1, [92].LeakTest.Basic.test_port := 1, [92].LeakTest.Basic.year := 26, [92].LeakTest.Basic.month := 6, [92].LeakTest.Basic.date := 4, [92].LeakTest.Basic.hour := 15, [92].LeakTest.Basic.minute := 7, [92].LeakTest.Basic.second := 3, [92].LeakTest.Basic.flags := 12, [92].LeakTest.Basic.Num_tests := 1, [92].LeakTest.Basic.test_elements.test_type := 66, [92].LeakTest.Basic.test_elements.test_eval := 1, [92].LeakTest.Basic.test_elements.num_elements := 16, [92].LeakTest.Detailed.unique_id := 42956, [92].LeakTest.Detailed.num_elements := 16, [92].LeakTest.Detailed.Test_Type := 66, [92].LeakTest.Detailed.element_data[0].Variable_code := 61, [92].LeakTest.Detailed.element_data[0].prec_code := 2, [92].LeakTest.Detailed.element_data[0].Unit_code := 60, [92].LeakTest.Detailed.element_data[0].result_measurement := 0.02514571, [92].LeakTest.Detailed.element_data[1].Variable_code := 28, [92].LeakTest.Detailed.element_data[1].prec_code := 3, [92].LeakTest.Detailed.element_data[1].Unit_code := 41, [92].LeakTest.Detailed.element_data[1].result_measurement := 0.00052619725, [92].LeakTest.Detailed.element_data[2].Variable_code := 13, [92].LeakTest.Detailed.element_data[2].prec_code := 3, [92].LeakTest.Detailed.element_data[2].Unit_code := 12, [92].LeakTest.Detailed.element_data[2].result_measurement := 5.231444, [92].LeakTest.Detailed.element_data[3].Variable_code := 75, [92].LeakTest.Detailed.element_data[3].prec_code := 2, [92].LeakTest.Detailed.element_data[3].Unit_code := 60, [92].LeakTest.Detailed.element_data[4].Variable_code := 60, [92].LeakTest.Detailed.element_data[4].prec_code := 2, [92].LeakTest.Detailed.element_data[4].Unit_code := 60, [92].LeakTest.Detailed.element_data[4].result_measurement := 0.020675361, [92].LeakTest.Detailed.element_data[5].Variable_code := 56, [92].LeakTest.Detailed.element_data[5].prec_code := 3, [92].LeakTest.Detailed.element_data[5].Unit_code := 41, [92].LeakTest.Detailed.element_data[5].result_measurement := 0.00017695129,
        [92].LeakTest.Detailed.element_data[6].Variable_code := 55, [92].LeakTest.Detailed.element_data[6].prec_code := 3, [92].LeakTest.Detailed.element_data[6].Unit_code := 12, [92].LeakTest.Detailed.element_data[6].result_measurement := 5.231444, [92].LeakTest.Detailed.element_data[7].Variable_code := 58, [92].LeakTest.Detailed.element_data[7].prec_code := 2, [92].LeakTest.Detailed.element_data[7].Unit_code := 60, [92].LeakTest.Detailed.element_data[7].result_measurement := -1.0002404, [92].LeakTest.Detailed.element_data[8].Variable_code := 59, [92].LeakTest.Detailed.element_data[8].prec_code := 2, [92].LeakTest.Detailed.element_data[8].Unit_code := 60, [92].LeakTest.Detailed.element_data[8].result_measurement := 1.0002404, [92].LeakTest.Detailed.element_data[9].Variable_code := 12, [92].LeakTest.Detailed.element_data[9].prec_code := 3, [92].LeakTest.Detailed.element_data[9].Unit_code := 12, [92].LeakTest.Detailed.element_data[9].result_measurement := 5.000001, [92].LeakTest.Detailed.element_data[10].Variable_code := 62, [92].LeakTest.Detailed.element_data[10].prec_code := 2, [92].LeakTest.Detailed.element_data[10].Unit_code := 60, [92].LeakTest.Detailed.element_data[10].result_measurement := 1.1298805, [92].LeakTest.Detailed.element_data[11].Variable_code := 21, [92].LeakTest.Detailed.element_data[11].prec_code := 3, [92].LeakTest.Detailed.element_data[11].Unit_code := 41, [92].LeakTest.Detailed.element_data[11].result_measurement := 4.656613e-06, [92].LeakTest.Detailed.element_data[12].Variable_code := 25, [92].LeakTest.Detailed.element_data[12].prec_code := 3, [92].LeakTest.Detailed.element_data[12].Unit_code := 41, [92].LeakTest.Detailed.element_data[12].result_measurement := 0.023245811, [92].LeakTest.Detailed.element_data[13].Variable_code := 216, [92].LeakTest.Detailed.element_data[13].prec_code := 3, [92].LeakTest.Detailed.element_data[13].Unit_code := 41, [92].LeakTest.Detailed.element_data[13].result_measurement := -3.7252903e-05, [92].LeakTest.Detailed.element_data[14].Variable_code := 218, [92].LeakTest.Detailed.element_data[14].prec_code := 3, [92].LeakTest.Detailed.element_data[14].Unit_code := 41, [92].LeakTest.Detailed.element_data[14].result_measurement := 0.011632219, [92].LeakTest.Detailed.element_data[15].Variable_code := 295, [92].LeakTest.Detailed.element_data[15].prec_code := 3, [92].LeakTest.Detailed.element_data[15].Unit_code := 12, [92].LeakTest.Detailed.element_data[15].result_measurement := 5.2328033, [93].Barcode := 'B252620969', [93].VolumeTest.UID := 41964, [93].VolumeTest.Basic.unique_id := 41964, [93].VolumeTest.Basic.channel_num := 1, [93].VolumeTest.Basic.program_num := 1, [93].VolumeTest.Basic.evaluation_code := 1, [93].VolumeTest.Basic.test_port := 1, [93].VolumeTest.Basic.year := 26, [93].VolumeTest.Basic.month := 6, [93].VolumeTest.Basic.date := 4, [93].VolumeTest.Basic.hour := 15, [93].VolumeTest.Basic.minute := 7, [93].VolumeTest.Basic.second := 46, [93].VolumeTest.Basic.flags := 12, [93].VolumeTest.Basic.Num_tests := 1, [93].VolumeTest.Basic.test_elements.test_type := 69, [93].VolumeTest.Basic.test_elements.test_eval := 1, [93].VolumeTest.Basic.test_elements.num_elements := 4, [93].VolumeTest.Detailed.unique_id := 41964, [93].VolumeTest.Detailed.num_elements := 4,
        [93].VolumeTest.Detailed.Test_Type := 69, [93].VolumeTest.Detailed.element_data[0].Variable_code := 245, [93].VolumeTest.Detailed.element_data[0].prec_code := 2, [93].VolumeTest.Detailed.element_data[0].Unit_code := 165, [93].VolumeTest.Detailed.element_data[0].result_measurement := 186.70047, [93].VolumeTest.Detailed.element_data[1].Variable_code := 13, [93].VolumeTest.Detailed.element_data[1].prec_code := 3, [93].VolumeTest.Detailed.element_data[1].Unit_code := 12, [93].VolumeTest.Detailed.element_data[1].result_measurement := 1.7814804, [93].VolumeTest.Detailed.element_data[2].Variable_code := 247, [93].VolumeTest.Detailed.element_data[2].prec_code := 3, [93].VolumeTest.Detailed.element_data[2].Unit_code := 12, [93].VolumeTest.Detailed.element_data[2].result_measurement := 5.1075125, [93].VolumeTest.Detailed.element_data[3].Variable_code := 295, [93].VolumeTest.Detailed.element_data[3].prec_code := 3, [93].VolumeTest.Detailed.element_data[3].Unit_code := 12, [93].VolumeTest.Detailed.element_data[3].result_measurement := 5.1079783, [93].LeakTest.UID := 41965, [93].LeakTest.Basic.unique_id := 41965, [93].LeakTest.Basic.channel_num := 1, [93].LeakTest.Basic.program_num := 2, [93].LeakTest.Basic.evaluation_code := 1, [93].LeakTest.Basic.test_port := 1, [93].LeakTest.Basic.year := 26, [93].LeakTest.Basic.month := 6, [93].LeakTest.Basic.date := 4, [93].LeakTest.Basic.hour := 15, [93].LeakTest.Basic.minute := 7, [93].LeakTest.Basic.second := 53, [93].LeakTest.Basic.flags := 12, [93].LeakTest.Basic.Num_tests := 1, [93].LeakTest.Basic.test_elements.test_type := 66, [93].LeakTest.Basic.test_elements.test_eval := 1, [93].LeakTest.Basic.test_elements.num_elements := 16, [93].LeakTest.Detailed.unique_id := 41965, [93].LeakTest.Detailed.num_elements := 16, [93].LeakTest.Detailed.Test_Type := 66, [93].LeakTest.Detailed.element_data[0].Variable_code := 61, [93].LeakTest.Detailed.element_data[0].prec_code := 2, [93].LeakTest.Detailed.element_data[0].Unit_code := 60, [93].LeakTest.Detailed.element_data[0].result_measurement := -0.06593764, [93].LeakTest.Detailed.element_data[1].Variable_code := 28, [93].LeakTest.Detailed.element_data[1].prec_code := 3, [93].LeakTest.Detailed.element_data[1].Unit_code := 41, [93].LeakTest.Detailed.element_data[1].result_measurement := 0.00029802322, [93].LeakTest.Detailed.element_data[2].Variable_code := 13, [93].LeakTest.Detailed.element_data[2].prec_code := 3, [93].LeakTest.Detailed.element_data[2].Unit_code := 12, [93].LeakTest.Detailed.element_data[2].result_measurement := 5.1366444, [93].LeakTest.Detailed.element_data[3].Variable_code := 75, [93].LeakTest.Detailed.element_data[3].prec_code := 2, [93].LeakTest.Detailed.element_data[3].Unit_code := 60, [93].LeakTest.Detailed.element_data[4].Variable_code := 60, [93].LeakTest.Detailed.element_data[4].prec_code := 2, [93].LeakTest.Detailed.element_data[4].Unit_code := 60, [93].LeakTest.Detailed.element_data[4].result_measurement := -0.06984919, [93].LeakTest.Detailed.element_data[5].Variable_code := 56, [93].LeakTest.Detailed.element_data[5].prec_code := 3, [93].LeakTest.Detailed.element_data[5].Unit_code := 41, [93].LeakTest.Detailed.element_data[5].result_measurement := 0.00021420419,
        [93].LeakTest.Detailed.element_data[6].Variable_code := 55, [93].LeakTest.Detailed.element_data[6].prec_code := 3, [93].LeakTest.Detailed.element_data[6].Unit_code := 12, [93].LeakTest.Detailed.element_data[6].result_measurement := 5.1366444, [93].LeakTest.Detailed.element_data[7].Variable_code := 58, [93].LeakTest.Detailed.element_data[7].prec_code := 2, [93].LeakTest.Detailed.element_data[7].Unit_code := 60, [93].LeakTest.Detailed.element_data[7].result_measurement := -1.0002404, [93].LeakTest.Detailed.element_data[8].Variable_code := 59, [93].LeakTest.Detailed.element_data[8].prec_code := 2, [93].LeakTest.Detailed.element_data[8].Unit_code := 60, [93].LeakTest.Detailed.element_data[8].result_measurement := 1.0002404, [93].LeakTest.Detailed.element_data[9].Variable_code := 12, [93].LeakTest.Detailed.element_data[9].prec_code := 3, [93].LeakTest.Detailed.element_data[9].Unit_code := 12, [93].LeakTest.Detailed.element_data[9].result_measurement := 5.000001, [93].LeakTest.Detailed.element_data[10].Variable_code := 62, [93].LeakTest.Detailed.element_data[10].prec_code := 2, [93].LeakTest.Detailed.element_data[10].Unit_code := 60, [93].LeakTest.Detailed.element_data[10].result_measurement := 1.1002644, [93].LeakTest.Detailed.element_data[11].Variable_code := 21, [93].LeakTest.Detailed.element_data[11].prec_code := 3, [93].LeakTest.Detailed.element_data[11].Unit_code := 41, [93].LeakTest.Detailed.element_data[11].result_measurement := 0.0015180558, [93].LeakTest.Detailed.element_data[12].Variable_code := 25, [93].LeakTest.Detailed.element_data[12].prec_code := 3, [93].LeakTest.Detailed.element_data[12].Unit_code := 41, [93].LeakTest.Detailed.element_data[12].result_measurement := 0.021727756, [93].LeakTest.Detailed.element_data[13].Variable_code := 216, [93].LeakTest.Detailed.element_data[13].prec_code := 3, [93].LeakTest.Detailed.element_data[13].Unit_code := 41, [93].LeakTest.Detailed.element_data[13].result_measurement := 0.00085681677, [93].LeakTest.Detailed.element_data[14].Variable_code := 218, [93].LeakTest.Detailed.element_data[14].prec_code := 3, [93].LeakTest.Detailed.element_data[14].Unit_code := 41, [93].LeakTest.Detailed.element_data[14].result_measurement := 0.01094304, [93].LeakTest.Detailed.element_data[15].Variable_code := 295, [93].LeakTest.Detailed.element_data[15].prec_code := 3, [93].LeakTest.Detailed.element_data[15].Unit_code := 12, [93].LeakTest.Detailed.element_data[15].result_measurement := 5.138372, [94].Barcode := 'B252620863', [94].VolumeTest.UID := 42958, [94].VolumeTest.Basic.unique_id := 42958, [94].VolumeTest.Basic.channel_num := 1, [94].VolumeTest.Basic.program_num := 1, [94].VolumeTest.Basic.evaluation_code := 1, [94].VolumeTest.Basic.test_port := 1, [94].VolumeTest.Basic.year := 26, [94].VolumeTest.Basic.month := 6, [94].VolumeTest.Basic.date := 4, [94].VolumeTest.Basic.hour := 15, [94].VolumeTest.Basic.minute := 8, [94].VolumeTest.Basic.second := 10, [94].VolumeTest.Basic.flags := 12, [94].VolumeTest.Basic.Num_tests := 1, [94].VolumeTest.Basic.test_elements.test_type := 69, [94].VolumeTest.Basic.test_elements.test_eval := 1, [94].VolumeTest.Basic.test_elements.num_elements := 4, [94].VolumeTest.Detailed.unique_id := 42958, [94].VolumeTest.Detailed.num_elements := 4,
        [94].VolumeTest.Detailed.Test_Type := 69, [94].VolumeTest.Detailed.element_data[0].Variable_code := 245, [94].VolumeTest.Detailed.element_data[0].prec_code := 2, [94].VolumeTest.Detailed.element_data[0].Unit_code := 165, [94].VolumeTest.Detailed.element_data[0].result_measurement := 188.24182, [94].VolumeTest.Detailed.element_data[1].Variable_code := 13, [94].VolumeTest.Detailed.element_data[1].prec_code := 3, [94].VolumeTest.Detailed.element_data[1].Unit_code := 12, [94].VolumeTest.Detailed.element_data[1].result_measurement := 1.8080837, [94].VolumeTest.Detailed.element_data[2].Variable_code := 247, [94].VolumeTest.Detailed.element_data[2].prec_code := 3, [94].VolumeTest.Detailed.element_data[2].Unit_code := 12, [94].VolumeTest.Detailed.element_data[2].result_measurement := 5.211653, [94].VolumeTest.Detailed.element_data[3].Variable_code := 295, [94].VolumeTest.Detailed.element_data[3].prec_code := 3, [94].VolumeTest.Detailed.element_data[3].Unit_code := 12, [94].VolumeTest.Detailed.element_data[3].result_measurement := 5.2136693, [94].LeakTest.UID := 42959, [94].LeakTest.Basic.unique_id := 42959, [94].LeakTest.Basic.channel_num := 1, [94].LeakTest.Basic.program_num := 2, [94].LeakTest.Basic.evaluation_code := 1, [94].LeakTest.Basic.test_port := 1, [94].LeakTest.Basic.year := 26, [94].LeakTest.Basic.month := 6, [94].LeakTest.Basic.date := 4, [94].LeakTest.Basic.hour := 15, [94].LeakTest.Basic.minute := 8, [94].LeakTest.Basic.second := 17, [94].LeakTest.Basic.flags := 12, [94].LeakTest.Basic.Num_tests := 1, [94].LeakTest.Basic.test_elements.test_type := 66, [94].LeakTest.Basic.test_elements.test_eval := 1, [94].LeakTest.Basic.test_elements.num_elements := 16, [94].LeakTest.Detailed.unique_id := 42959, [94].LeakTest.Detailed.num_elements := 16, [94].LeakTest.Detailed.Test_Type := 66, [94].LeakTest.Detailed.element_data[0].Variable_code := 61, [94].LeakTest.Detailed.element_data[0].prec_code := 2, [94].LeakTest.Detailed.element_data[0].Unit_code := 60, [94].LeakTest.Detailed.element_data[0].result_measurement := -999.0, [94].LeakTest.Detailed.element_data[1].Variable_code := 28, [94].LeakTest.Detailed.element_data[1].prec_code := 3, [94].LeakTest.Detailed.element_data[1].Unit_code := 41, [94].LeakTest.Detailed.element_data[1].result_measurement := -4.656613e-06, [94].LeakTest.Detailed.element_data[2].Variable_code := 13, [94].LeakTest.Detailed.element_data[2].prec_code := 3, [94].LeakTest.Detailed.element_data[2].Unit_code := 12, [94].LeakTest.Detailed.element_data[2].result_measurement := 5.2301817, [94].LeakTest.Detailed.element_data[3].Variable_code := 75, [94].LeakTest.Detailed.element_data[3].prec_code := 2, [94].LeakTest.Detailed.element_data[3].Unit_code := 60, [94].LeakTest.Detailed.element_data[4].Variable_code := 60, [94].LeakTest.Detailed.element_data[4].prec_code := 2, [94].LeakTest.Detailed.element_data[4].Unit_code := 60, [94].LeakTest.Detailed.element_data[4].result_measurement := 0.0027939677, [94].LeakTest.Detailed.element_data[5].Variable_code := 56, [94].LeakTest.Detailed.element_data[5].prec_code := 3, [94].LeakTest.Detailed.element_data[5].Unit_code := 41, [94].LeakTest.Detailed.element_data[5].result_measurement := -4.656613e-06,
        [94].LeakTest.Detailed.element_data[6].Variable_code := 55, [94].LeakTest.Detailed.element_data[6].prec_code := 3, [94].LeakTest.Detailed.element_data[6].Unit_code := 12, [94].LeakTest.Detailed.element_data[6].result_measurement := 5.2301817, [94].LeakTest.Detailed.element_data[7].Variable_code := 58, [94].LeakTest.Detailed.element_data[7].prec_code := 2, [94].LeakTest.Detailed.element_data[7].Unit_code := 60, [94].LeakTest.Detailed.element_data[7].result_measurement := -1.0002404, [94].LeakTest.Detailed.element_data[8].Variable_code := 59, [94].LeakTest.Detailed.element_data[8].prec_code := 2, [94].LeakTest.Detailed.element_data[8].Unit_code := 60, [94].LeakTest.Detailed.element_data[8].result_measurement := 1.0002404, [94].LeakTest.Detailed.element_data[9].Variable_code := 12, [94].LeakTest.Detailed.element_data[9].prec_code := 3, [94].LeakTest.Detailed.element_data[9].Unit_code := 12, [94].LeakTest.Detailed.element_data[9].result_measurement := 5.000001, [94].LeakTest.Detailed.element_data[10].Variable_code := 62, [94].LeakTest.Detailed.element_data[10].prec_code := 2, [94].LeakTest.Detailed.element_data[10].Unit_code := 60, [94].LeakTest.Detailed.element_data[10].result_measurement := 1.1298805, [94].LeakTest.Detailed.element_data[11].Variable_code := 21, [94].LeakTest.Detailed.element_data[11].prec_code := 3, [94].LeakTest.Detailed.element_data[11].Unit_code := 41, [94].LeakTest.Detailed.element_data[11].result_measurement := 4.656613e-06, [94].LeakTest.Detailed.element_data[12].Variable_code := 25, [94].LeakTest.Detailed.element_data[12].prec_code := 3, [94].LeakTest.Detailed.element_data[12].Unit_code := 41, [94].LeakTest.Detailed.element_data[12].result_measurement := 0.023245811, [94].LeakTest.Detailed.element_data[13].Variable_code := 216, [94].LeakTest.Detailed.element_data[13].prec_code := 3, [94].LeakTest.Detailed.element_data[13].Unit_code := 41, [94].LeakTest.Detailed.element_data[13].result_measurement := -3.7252903e-05, [94].LeakTest.Detailed.element_data[14].Variable_code := 218, [94].LeakTest.Detailed.element_data[14].prec_code := 3, [94].LeakTest.Detailed.element_data[14].Unit_code := 41, [94].LeakTest.Detailed.element_data[14].result_measurement := 0.011632219, [94].LeakTest.Detailed.element_data[15].Variable_code := 295, [94].LeakTest.Detailed.element_data[15].prec_code := 3, [94].LeakTest.Detailed.element_data[15].Unit_code := 12, [94].LeakTest.Detailed.element_data[15].result_measurement := 5.23197, [95].Barcode := 'B252620969', [95].VolumeTest.UID := 42961, [95].VolumeTest.Basic.unique_id := 42961, [95].VolumeTest.Basic.channel_num := 1, [95].VolumeTest.Basic.program_num := 1, [95].VolumeTest.Basic.evaluation_code := 1, [95].VolumeTest.Basic.test_port := 1, [95].VolumeTest.Basic.year := 26, [95].VolumeTest.Basic.month := 6, [95].VolumeTest.Basic.date := 4, [95].VolumeTest.Basic.hour := 15, [95].VolumeTest.Basic.minute := 9, [95].VolumeTest.Basic.second := 40, [95].VolumeTest.Basic.flags := 12, [95].VolumeTest.Basic.Num_tests := 1, [95].VolumeTest.Basic.test_elements.test_type := 69, [95].VolumeTest.Basic.test_elements.test_eval := 1, [95].VolumeTest.Basic.test_elements.num_elements := 4, [95].VolumeTest.Detailed.unique_id := 42961, [95].VolumeTest.Detailed.num_elements := 4,
